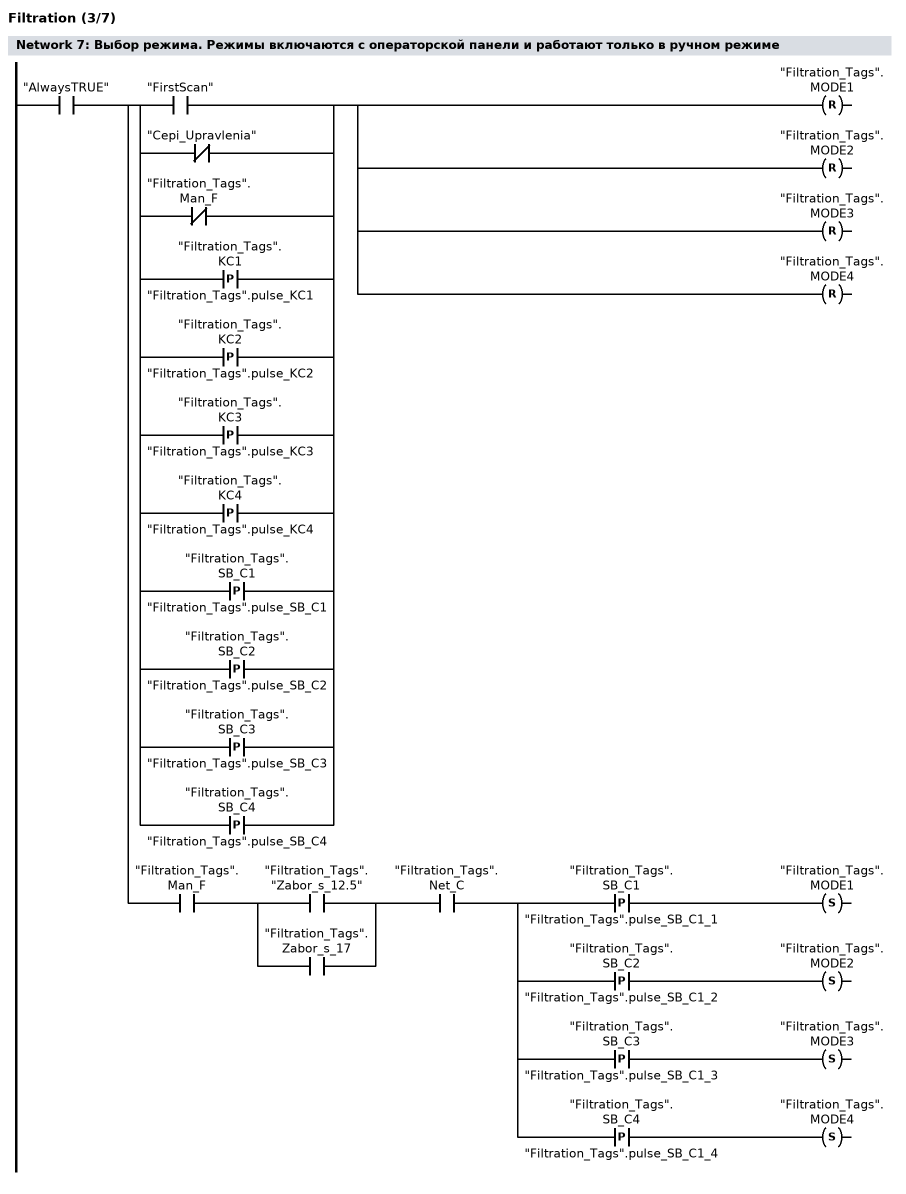
   RUNG wire#powerrail
      Contact( "AlwaysTRUE" )
      wire#w1
      Contact( "FirstScan" )
      wire#w2
      R_Coil( "Filtration_Tags".MODE1 )
   END_RUNG
   RUNG wire#w1
      I_Contact( "Cepi_Upravlenia" )
   END_RUNG wire#w2
   RUNG wire#w1
      I_Contact( "Filtration_Tags".Man_F )
   END_RUNG wire#w2
   RUNG wire#w1
      P_Contact(operand := "Filtration_Tags".KC1, bit := "Filtration_Tags".pulse_KC1)
   END_RUNG wire#w2
   RUNG wire#w1
      P_Contact(operand := "Filtration_Tags".KC2, bit := "Filtration_Tags".pulse_KC2)
   END_RUNG wire#w2
   RUNG wire#w1
      P_Contact(operand := "Filtration_Tags".KC3, bit := "Filtration_Tags".pulse_KC3)
   END_RUNG wire#w2
   RUNG wire#w1
      P_Contact(operand := "Filtration_Tags".KC4, bit := "Filtration_Tags".pulse_KC4)
   END_RUNG wire#w2
   RUNG wire#w1
      P_Contact(operand := "Filtration_Tags".SB_C1, bit := "Filtration_Tags".pulse_SB_C1)
   END_RUNG wire#w2
   RUNG wire#w1
      P_Contact(operand := "Filtration_Tags".SB_C2, bit := "Filtration_Tags".pulse_SB_C2)
   END_RUNG wire#w2
   RUNG wire#w1
      P_Contact(operand := "Filtration_Tags".SB_C3, bit := "Filtration_Tags".pulse_SB_C3)
   END_RUNG wire#w2
   RUNG wire#w1
      P_Contact(operand := "Filtration_Tags".SB_C4, bit := "Filtration_Tags".pulse_SB_C4)
   END_RUNG wire#w2
   RUNG wire#w2
      R_Coil( "Filtration_Tags".MODE2 )
   END_RUNG
   RUNG wire#w2
      R_Coil( "Filtration_Tags".MODE3 )
   END_RUNG
   RUNG wire#w2
      R_Coil( "Filtration_Tags".MODE4 )
   END_RUNG
   RUNG wire#w1
      Contact( "Filtration_Tags".Man_F )
      wire#w3
      Contact( "Filtration_Tags"."Zabor_s_12.5" )
      wire#w4
      Contact( "Filtration_Tags".Net_C )
      wire#w5
      P_Contact(operand := "Filtration_Tags".SB_C1, bit := "Filtration_Tags".pulse_SB_C1_1)
      S_Coil( "Filtration_Tags".MODE1 )
   END_RUNG
   RUNG wire#w3
      Contact( "Filtration_Tags".Zabor_s_17 )
   END_RUNG wire#w4
   RUNG wire#w5
      P_Contact(operand := "Filtration_Tags".SB_C2, bit := "Filtration_Tags".pulse_SB_C1_2)
      S_Coil( "Filtration_Tags".MODE2 )
   END_RUNG
   RUNG wire#w5
      P_Contact(operand := "Filtration_Tags".SB_C3, bit := "Filtration_Tags".pulse_SB_C1_3)
      S_Coil( "Filtration_Tags".MODE3 )
   END_RUNG
   RUNG wire#w5
      P_Contact(operand := "Filtration_Tags".SB_C4, bit := "Filtration_Tags".pulse_SB_C1_4)
      S_Coil( "Filtration_Tags".MODE4 )
   END_RUNG
   // the same network as SCL:
   #_w1 := "AlwaysTRUE" AND "Filtration_Tags".KC1 AND NOT "Filtration_Tags".pulse_KC1;   // rising edge of "Filtration_Tags".KC1
   "Filtration_Tags".pulse_KC1 := "Filtration_Tags".KC1;
   #_w2 := "AlwaysTRUE" AND "Filtration_Tags".KC2 AND NOT "Filtration_Tags".pulse_KC2;   // rising edge of "Filtration_Tags".KC2
   "Filtration_Tags".pulse_KC2 := "Filtration_Tags".KC2;
   #_w3 := "AlwaysTRUE" AND "Filtration_Tags".KC3 AND NOT "Filtration_Tags".pulse_KC3;   // rising edge of "Filtration_Tags".KC3
   "Filtration_Tags".pulse_KC3 := "Filtration_Tags".KC3;
   #_w4 := "AlwaysTRUE" AND "Filtration_Tags".KC4 AND NOT "Filtration_Tags".pulse_KC4;   // rising edge of "Filtration_Tags".KC4
   "Filtration_Tags".pulse_KC4 := "Filtration_Tags".KC4;
   #_w5 := "AlwaysTRUE" AND "Filtration_Tags".SB_C1 AND NOT "Filtration_Tags".pulse_SB_C1;   // rising edge of "Filtration_Tags".SB_C1
   "Filtration_Tags".pulse_SB_C1 := "Filtration_Tags".SB_C1;
   #_w6 := "AlwaysTRUE" AND "Filtration_Tags".SB_C2 AND NOT "Filtration_Tags".pulse_SB_C2;   // rising edge of "Filtration_Tags".SB_C2
   "Filtration_Tags".pulse_SB_C2 := "Filtration_Tags".SB_C2;
   #_w7 := "AlwaysTRUE" AND "Filtration_Tags".SB_C3 AND NOT "Filtration_Tags".pulse_SB_C3;   // rising edge of "Filtration_Tags".SB_C3
   "Filtration_Tags".pulse_SB_C3 := "Filtration_Tags".SB_C3;
   #_w8 := "AlwaysTRUE" AND "Filtration_Tags".SB_C4 AND NOT "Filtration_Tags".pulse_SB_C4;   // rising edge of "Filtration_Tags".SB_C4
   "Filtration_Tags".pulse_SB_C4 := "Filtration_Tags".SB_C4;
   IF ("AlwaysTRUE" AND ("FirstScan" OR NOT "Cepi_Upravlenia" OR NOT "Filtration_Tags".Man_F)) OR #_w1 OR #_w2 OR #_w3 OR #_w4 OR #_w5 OR #_w6 OR #_w7 OR #_w8 THEN
       "Filtration_Tags".MODE1 := FALSE;
       "Filtration_Tags".MODE2 := FALSE;
       "Filtration_Tags".MODE3 := FALSE;
       "Filtration_Tags".MODE4 := FALSE;
   END_IF;
   #_w9 := "AlwaysTRUE" AND "Filtration_Tags".Man_F AND ("Filtration_Tags"."Zabor_s_12.5" OR "Filtration_Tags".Zabor_s_17) AND "Filtration_Tags".Net_C;
   #_w10 := #_w9 AND "Filtration_Tags".SB_C1 AND NOT "Filtration_Tags".pulse_SB_C1_1;   // rising edge of "Filtration_Tags".SB_C1
   "Filtration_Tags".pulse_SB_C1_1 := "Filtration_Tags".SB_C1;
   IF #_w10 THEN "Filtration_Tags".MODE1 := TRUE; END_IF;
   #_w11 := #_w9 AND "Filtration_Tags".SB_C2 AND NOT "Filtration_Tags".pulse_SB_C1_2;   // rising edge of "Filtration_Tags".SB_C2
   "Filtration_Tags".pulse_SB_C1_2 := "Filtration_Tags".SB_C2;
   IF #_w11 THEN "Filtration_Tags".MODE2 := TRUE; END_IF;
   #_w12 := #_w9 AND "Filtration_Tags".SB_C3 AND NOT "Filtration_Tags".pulse_SB_C1_3;   // rising edge of "Filtration_Tags".SB_C3
   "Filtration_Tags".pulse_SB_C1_3 := "Filtration_Tags".SB_C3;
   IF #_w12 THEN "Filtration_Tags".MODE3 := TRUE; END_IF;
   #_w13 := #_w9 AND "Filtration_Tags".SB_C4 AND NOT "Filtration_Tags".pulse_SB_C1_4;   // rising edge of "Filtration_Tags".SB_C4
   "Filtration_Tags".pulse_SB_C1_4 := "Filtration_Tags".SB_C4;
   IF #_w13 THEN "Filtration_Tags".MODE4 := TRUE; END_IF;
END_REGION

REGION Network 8: Цикл 1. Заправка фильтра
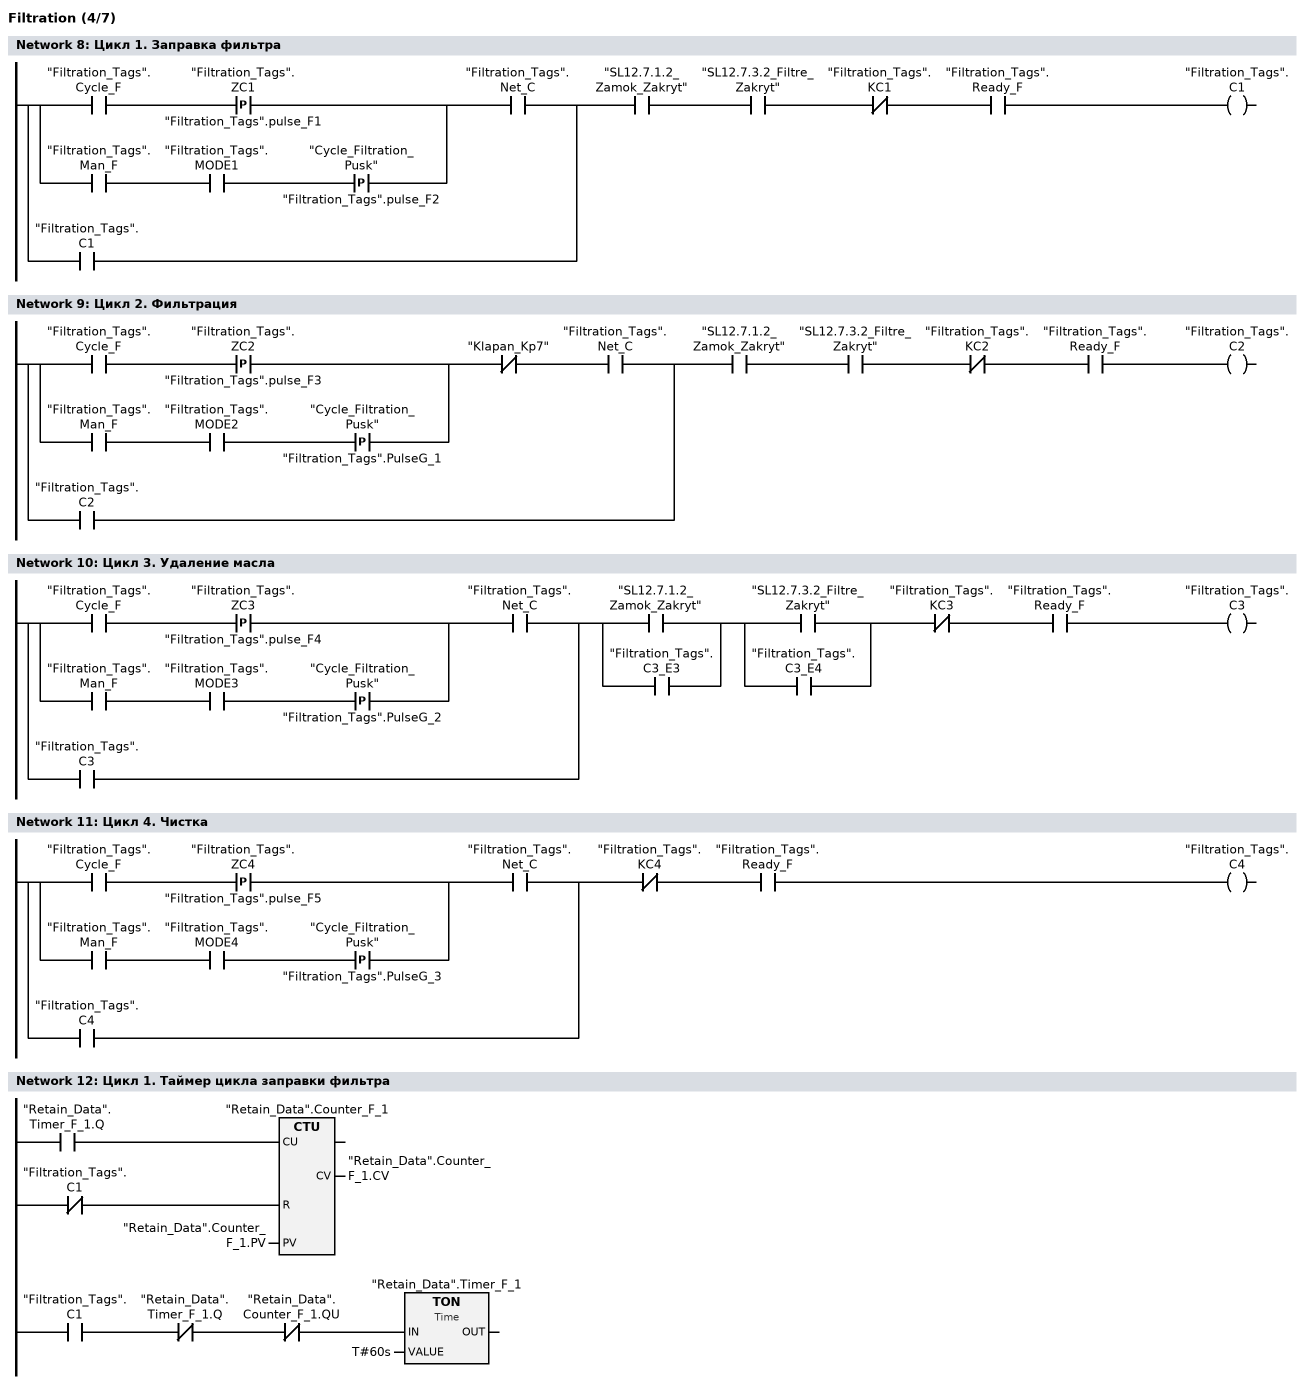
   RUNG wire#powerrail
      Contact( "Filtration_Tags".Cycle_F )
      P_Contact(operand := "Filtration_Tags".ZC1, bit := "Filtration_Tags".pulse_F1)
      wire#w1
      Contact( "Filtration_Tags".Net_C )
      wire#w2
      Contact( "SL12.7.1.2_Zamok_Zakryt" )
      Contact( "SL12.7.3.2_Filtre_Zakryt" )
      I_Contact( "Filtration_Tags".KC1 )
      Contact( "Filtration_Tags".Ready_F )
      Coil( "Filtration_Tags".C1 )
   END_RUNG
   RUNG wire#powerrail
      Contact( "Filtration_Tags".Man_F )
      Contact( "Filtration_Tags".MODE1 )
      P_Contact(operand := "Cycle_Filtration_Pusk", bit := "Filtration_Tags".pulse_F2)
   END_RUNG wire#w1
   RUNG wire#powerrail
      Contact( "Filtration_Tags".C1 )
   END_RUNG wire#w2
   // the same network as SCL:
   #_w1 := "Filtration_Tags".Cycle_F AND "Filtration_Tags".ZC1 AND NOT "Filtration_Tags".pulse_F1;   // rising edge of "Filtration_Tags".ZC1
   "Filtration_Tags".pulse_F1 := "Filtration_Tags".ZC1;
   #_w2 := "Filtration_Tags".Man_F AND "Filtration_Tags".MODE1 AND "Cycle_Filtration_Pusk" AND NOT "Filtration_Tags".pulse_F2;   // rising edge of "Cycle_Filtration_Pusk"
   "Filtration_Tags".pulse_F2 := "Cycle_Filtration_Pusk";
   "Filtration_Tags".C1 := (((#_w1 OR #_w2) AND "Filtration_Tags".Net_C) OR "Filtration_Tags".C1) AND "SL12.7.1.2_Zamok_Zakryt" AND "SL12.7.3.2_Filtre_Zakryt" AND NOT "Filtration_Tags".KC1 AND "Filtration_Tags".Ready_F;
END_REGION

REGION Network 9: Цикл 2. Фильтрация
   RUNG wire#powerrail
      Contact( "Filtration_Tags".Cycle_F )
      P_Contact(operand := "Filtration_Tags".ZC2, bit := "Filtration_Tags".pulse_F3)
      wire#w1
      I_Contact( "Klapan_Kp7" )
      Contact( "Filtration_Tags".Net_C )
      wire#w2
      Contact( "SL12.7.1.2_Zamok_Zakryt" )
      Contact( "SL12.7.3.2_Filtre_Zakryt" )
      I_Contact( "Filtration_Tags".KC2 )
      Contact( "Filtration_Tags".Ready_F )
      Coil( "Filtration_Tags".C2 )
   END_RUNG
   RUNG wire#powerrail
      Contact( "Filtration_Tags".Man_F )
      Contact( "Filtration_Tags".MODE2 )
      P_Contact(operand := "Cycle_Filtration_Pusk", bit := "Filtration_Tags".PulseG_1)
   END_RUNG wire#w1
   RUNG wire#powerrail
      Contact( "Filtration_Tags".C2 )
   END_RUNG wire#w2
   // the same network as SCL:
   #_w1 := "Filtration_Tags".Cycle_F AND "Filtration_Tags".ZC2 AND NOT "Filtration_Tags".pulse_F3;   // rising edge of "Filtration_Tags".ZC2
   "Filtration_Tags".pulse_F3 := "Filtration_Tags".ZC2;
   #_w2 := "Filtration_Tags".Man_F AND "Filtration_Tags".MODE2 AND "Cycle_Filtration_Pusk" AND NOT "Filtration_Tags".PulseG_1;   // rising edge of "Cycle_Filtration_Pusk"
   "Filtration_Tags".PulseG_1 := "Cycle_Filtration_Pusk";
   "Filtration_Tags".C2 := (((#_w1 OR #_w2) AND NOT "Klapan_Kp7" AND "Filtration_Tags".Net_C) OR "Filtration_Tags".C2) AND "SL12.7.1.2_Zamok_Zakryt" AND "SL12.7.3.2_Filtre_Zakryt" AND NOT "Filtration_Tags".KC2 AND "Filtration_Tags".Ready_F;
END_REGION

REGION Network 10: Цикл 3. Удаление масла
   RUNG wire#powerrail
      Contact( "Filtration_Tags".Cycle_F )
      P_Contact(operand := "Filtration_Tags".ZC3, bit := "Filtration_Tags".pulse_F4)
      wire#w1
      Contact( "Filtration_Tags".Net_C )
      wire#w2
      Contact( "SL12.7.1.2_Zamok_Zakryt" )
      wire#w3
      Contact( "SL12.7.3.2_Filtre_Zakryt" )
      wire#w4
      I_Contact( "Filtration_Tags".KC3 )
      Contact( "Filtration_Tags".Ready_F )
      Coil( "Filtration_Tags".C3 )
   END_RUNG
   RUNG wire#powerrail
      Contact( "Filtration_Tags".Man_F )
      Contact( "Filtration_Tags".MODE3 )
      P_Contact(operand := "Cycle_Filtration_Pusk", bit := "Filtration_Tags".PulseG_2)
   END_RUNG wire#w1
   RUNG wire#powerrail
      Contact( "Filtration_Tags".C3 )
   END_RUNG wire#w2
   RUNG wire#w2
      Contact( "Filtration_Tags".C3_E3 )
   END_RUNG wire#w3
   RUNG wire#w3
      Contact( "Filtration_Tags".C3_E4 )
   END_RUNG wire#w4
   // the same network as SCL:
   #_w1 := "Filtration_Tags".Cycle_F AND "Filtration_Tags".ZC3 AND NOT "Filtration_Tags".pulse_F4;   // rising edge of "Filtration_Tags".ZC3
   "Filtration_Tags".pulse_F4 := "Filtration_Tags".ZC3;
   #_w2 := "Filtration_Tags".Man_F AND "Filtration_Tags".MODE3 AND "Cycle_Filtration_Pusk" AND NOT "Filtration_Tags".PulseG_2;   // rising edge of "Cycle_Filtration_Pusk"
   "Filtration_Tags".PulseG_2 := "Cycle_Filtration_Pusk";
   "Filtration_Tags".C3 := (((#_w1 OR #_w2) AND "Filtration_Tags".Net_C) OR "Filtration_Tags".C3) AND ("SL12.7.1.2_Zamok_Zakryt" OR "Filtration_Tags".C3_E3) AND ("SL12.7.3.2_Filtre_Zakryt" OR "Filtration_Tags".C3_E4) AND NOT "Filtration_Tags".KC3 AND "Filtration_Tags".Ready_F;
END_REGION

REGION Network 11: Цикл 4. Чистка
   RUNG wire#powerrail
      Contact( "Filtration_Tags".Cycle_F )
      P_Contact(operand := "Filtration_Tags".ZC4, bit := "Filtration_Tags".pulse_F5)
      wire#w1
      Contact( "Filtration_Tags".Net_C )
      wire#w2
      I_Contact( "Filtration_Tags".KC4 )
      Contact( "Filtration_Tags".Ready_F )
      Coil( "Filtration_Tags".C4 )
   END_RUNG
   RUNG wire#powerrail
      Contact( "Filtration_Tags".Man_F )
      Contact( "Filtration_Tags".MODE4 )
      P_Contact(operand := "Cycle_Filtration_Pusk", bit := "Filtration_Tags".PulseG_3)
   END_RUNG wire#w1
   RUNG wire#powerrail
      Contact( "Filtration_Tags".C4 )
   END_RUNG wire#w2
   // the same network as SCL:
   #_w1 := "Filtration_Tags".Cycle_F AND "Filtration_Tags".ZC4 AND NOT "Filtration_Tags".pulse_F5;   // rising edge of "Filtration_Tags".ZC4
   "Filtration_Tags".pulse_F5 := "Filtration_Tags".ZC4;
   #_w2 := "Filtration_Tags".Man_F AND "Filtration_Tags".MODE4 AND "Cycle_Filtration_Pusk" AND NOT "Filtration_Tags".PulseG_3;   // rising edge of "Cycle_Filtration_Pusk"
   "Filtration_Tags".PulseG_3 := "Cycle_Filtration_Pusk";
   "Filtration_Tags".C4 := (((#_w1 OR #_w2) AND "Filtration_Tags".Net_C) OR "Filtration_Tags".C4) AND NOT "Filtration_Tags".KC4 AND "Filtration_Tags".Ready_F;
END_REGION

REGION Network 12: Цикл 1. Таймер цикла заправки фильтра
   "Retain_Data".Counter_F_1.CTU(CU := "Retain_Data".Timer_F_1.Q,
                           R := NOT "Filtration_Tags".C1,
                           PV := "Retain_Data".Counter_F_1.PV,
                           CV => "Retain_Data".Counter_F_1.CV);
   "Retain_Data".Timer_F_1.TON(IN := "Filtration_Tags".C1 AND NOT "Retain_Data".Timer_F_1.Q AND NOT "Retain_Data".Counter_F_1.QU, PT := T#60s);   // TON coil
END_REGION

REGION Network 13: Цикл 1. Таймер работы клапана декомпрессии Кд
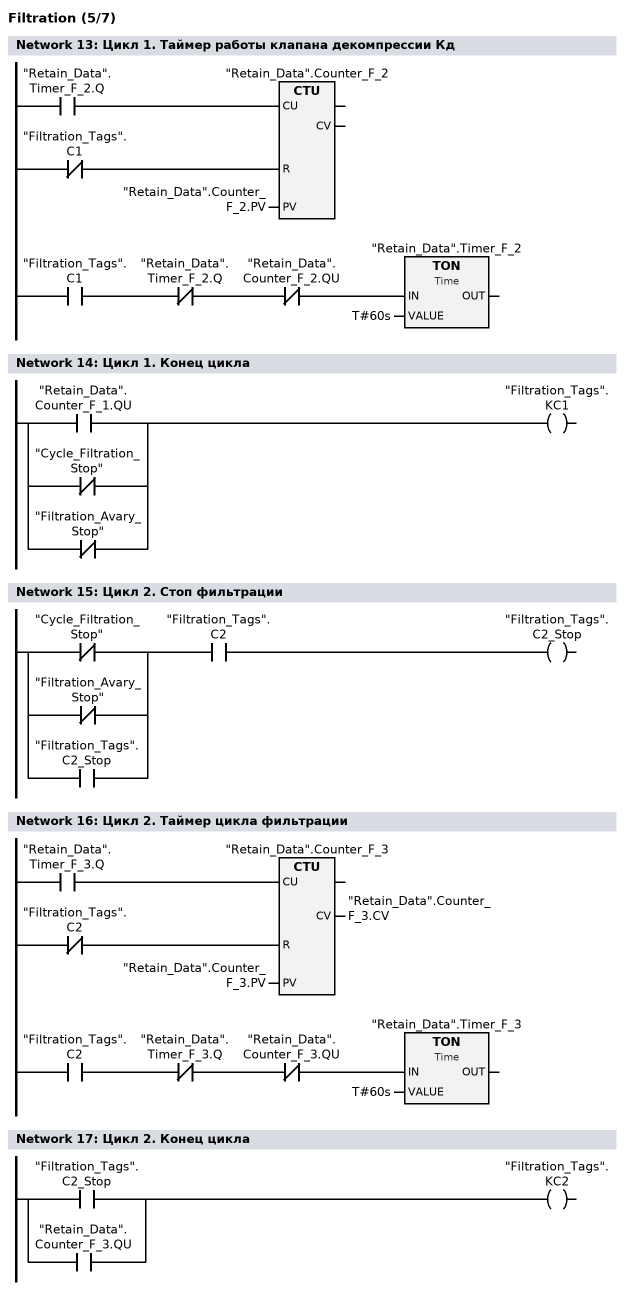
   "Retain_Data".Counter_F_2.CTU(CU := "Retain_Data".Timer_F_2.Q,
                           R := NOT "Filtration_Tags".C1,
                           PV := "Retain_Data".Counter_F_2.PV);
   "Retain_Data".Timer_F_2.TON(IN := "Filtration_Tags".C1 AND NOT "Retain_Data".Timer_F_2.Q AND NOT "Retain_Data".Counter_F_2.QU, PT := T#60s);   // TON coil
END_REGION

REGION Network 14: Цикл 1. Конец цикла
   RUNG wire#powerrail
      Contact( "Retain_Data".Counter_F_1.QU )
      wire#w1
      Coil( "Filtration_Tags".KC1 )
   END_RUNG
   RUNG wire#powerrail
      I_Contact( "Cycle_Filtration_Stop" )
   END_RUNG wire#w1
   RUNG wire#powerrail
      I_Contact( "Filtration_Avary_Stop" )
   END_RUNG wire#w1
   // the same network as SCL:
   "Filtration_Tags".KC1 := "Retain_Data".Counter_F_1.QU OR NOT "Cycle_Filtration_Stop" OR NOT "Filtration_Avary_Stop";
END_REGION

REGION Network 15: Цикл 2. Стоп фильтрации
   RUNG wire#powerrail
      I_Contact( "Cycle_Filtration_Stop" )
      wire#w1
      Contact( "Filtration_Tags".C2 )
      Coil( "Filtration_Tags".C2_Stop )
   END_RUNG
   RUNG wire#powerrail
      I_Contact( "Filtration_Avary_Stop" )
   END_RUNG wire#w1
   RUNG wire#powerrail
      Contact( "Filtration_Tags".C2_Stop )
   END_RUNG wire#w1
   // the same network as SCL:
   "Filtration_Tags".C2_Stop := (NOT "Cycle_Filtration_Stop" OR NOT "Filtration_Avary_Stop" OR "Filtration_Tags".C2_Stop) AND "Filtration_Tags".C2;
END_REGION

REGION Network 16: Цикл 2. Таймер цикла фильтрации
   "Retain_Data".Counter_F_3.CTU(CU := "Retain_Data".Timer_F_3.Q,
                           R := NOT "Filtration_Tags".C2,
                           PV := "Retain_Data".Counter_F_3.PV,
                           CV => "Retain_Data".Counter_F_3.CV);
   "Retain_Data".Timer_F_3.TON(IN := "Filtration_Tags".C2 AND NOT "Retain_Data".Timer_F_3.Q AND NOT "Retain_Data".Counter_F_3.QU, PT := T#60s);   // TON coil
END_REGION

REGION Network 17: Цикл 2. Конец цикла
   RUNG wire#powerrail
      Contact( "Filtration_Tags".C2_Stop )
      wire#w1
      Coil( "Filtration_Tags".KC2 )
   END_RUNG
   RUNG wire#powerrail
      Contact( "Retain_Data".Counter_F_3.QU )
   END_RUNG wire#w1
   // the same network as SCL:
   "Filtration_Tags".KC2 := "Filtration_Tags".C2_Stop OR "Retain_Data".Counter_F_3.QU;
END_REGION

REGION Network 18: Цикл 3. Циклограмма удаления масла
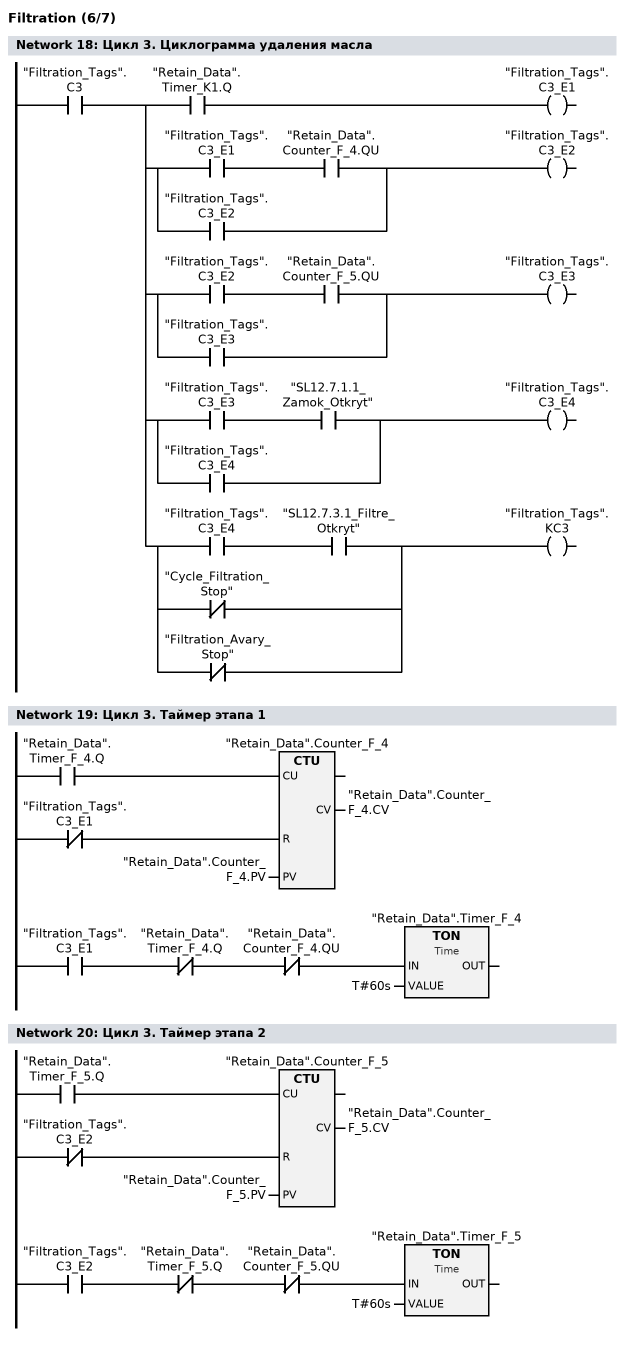
   RUNG wire#powerrail
      Contact( "Filtration_Tags".C3 )
      wire#w1
      Contact( "Retain_Data".Timer_K1.Q )
      Coil( "Filtration_Tags".C3_E1 )
   END_RUNG
   RUNG wire#w1
      Contact( "Filtration_Tags".C3_E1 )
      Contact( "Retain_Data".Counter_F_4.QU )
      wire#w2
      Coil( "Filtration_Tags".C3_E2 )
   END_RUNG
   RUNG wire#w1
      Contact( "Filtration_Tags".C3_E2 )
   END_RUNG wire#w2
   RUNG wire#w1
      Contact( "Filtration_Tags".C3_E2 )
      Contact( "Retain_Data".Counter_F_5.QU )
      wire#w3
      Coil( "Filtration_Tags".C3_E3 )
   END_RUNG
   RUNG wire#w1
      Contact( "Filtration_Tags".C3_E3 )
   END_RUNG wire#w3
   RUNG wire#w1
      Contact( "Filtration_Tags".C3_E3 )
      Contact( "SL12.7.1.1_Zamok_Otkryt" )
      wire#w4
      Coil( "Filtration_Tags".C3_E4 )
   END_RUNG
   RUNG wire#w1
      Contact( "Filtration_Tags".C3_E4 )
   END_RUNG wire#w4
   RUNG wire#w1
      Contact( "Filtration_Tags".C3_E4 )
      Contact( "SL12.7.3.1_Filtre_Otkryt" )
      wire#w5
      Coil( "Filtration_Tags".KC3 )
   END_RUNG
   RUNG wire#w1
      I_Contact( "Cycle_Filtration_Stop" )
   END_RUNG wire#w5
   RUNG wire#w1
      I_Contact( "Filtration_Avary_Stop" )
   END_RUNG wire#w5
   // the same network as SCL:
   "Filtration_Tags".C3_E1 := "Filtration_Tags".C3 AND "Retain_Data".Timer_K1.Q;
   "Filtration_Tags".C3_E2 := "Filtration_Tags".C3 AND (("Filtration_Tags".C3_E1 AND "Retain_Data".Counter_F_4.QU) OR "Filtration_Tags".C3_E2);
   "Filtration_Tags".C3_E3 := "Filtration_Tags".C3 AND (("Filtration_Tags".C3_E2 AND "Retain_Data".Counter_F_5.QU) OR "Filtration_Tags".C3_E3);
   "Filtration_Tags".C3_E4 := "Filtration_Tags".C3 AND (("Filtration_Tags".C3_E3 AND "SL12.7.1.1_Zamok_Otkryt") OR "Filtration_Tags".C3_E4);
   "Filtration_Tags".KC3 := "Filtration_Tags".C3 AND (("Filtration_Tags".C3_E4 AND "SL12.7.3.1_Filtre_Otkryt") OR NOT "Cycle_Filtration_Stop" OR NOT "Filtration_Avary_Stop");
END_REGION

REGION Network 19: Цикл 3. Таймер этапа 1
   "Retain_Data".Counter_F_4.CTU(CU := "Retain_Data".Timer_F_4.Q,
                           R := NOT "Filtration_Tags".C3_E1,
                           PV := "Retain_Data".Counter_F_4.PV,
                           CV => "Retain_Data".Counter_F_4.CV);
   "Retain_Data".Timer_F_4.TON(IN := "Filtration_Tags".C3_E1 AND NOT "Retain_Data".Timer_F_4.Q AND NOT "Retain_Data".Counter_F_4.QU, PT := T#60s);   // TON coil
END_REGION

REGION Network 20: Цикл 3. Таймер этапа 2
   "Retain_Data".Counter_F_5.CTU(CU := "Retain_Data".Timer_F_5.Q,
                           R := NOT "Filtration_Tags".C3_E2,
                           PV := "Retain_Data".Counter_F_5.PV,
                           CV => "Retain_Data".Counter_F_5.CV);
   "Retain_Data".Timer_F_5.TON(IN := "Filtration_Tags".C3_E2 AND NOT "Retain_Data".Timer_F_5.Q AND NOT "Retain_Data".Counter_F_5.QU, PT := T#60s);   // TON coil
END_REGION

REGION Network 21: Цикл 4. Циклограмма чистки
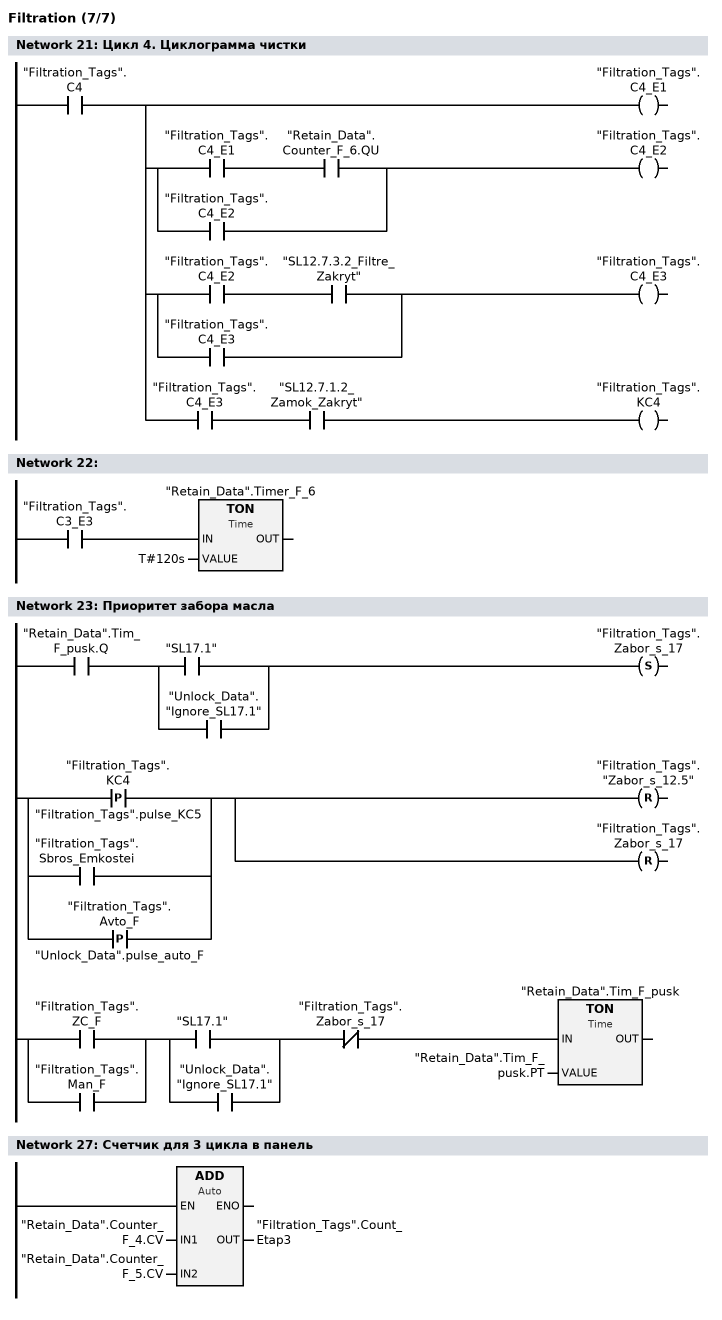
   RUNG wire#powerrail
      Contact( "Filtration_Tags".C4 )
      wire#w1
      Coil( "Filtration_Tags".C4_E1 )
   END_RUNG
   RUNG wire#w1
      Contact( "Filtration_Tags".C4_E1 )
      Contact( "Retain_Data".Counter_F_6.QU )
      wire#w2
      Coil( "Filtration_Tags".C4_E2 )
   END_RUNG
   RUNG wire#w1
      Contact( "Filtration_Tags".C4_E2 )
   END_RUNG wire#w2
   RUNG wire#w1
      Contact( "Filtration_Tags".C4_E2 )
      Contact( "SL12.7.3.2_Filtre_Zakryt" )
      wire#w3
      Coil( "Filtration_Tags".C4_E3 )
   END_RUNG
   RUNG wire#w1
      Contact( "Filtration_Tags".C4_E3 )
   END_RUNG wire#w3
   RUNG wire#w1
      Contact( "Filtration_Tags".C4_E3 )
      Contact( "SL12.7.1.2_Zamok_Zakryt" )
      Coil( "Filtration_Tags".KC4 )
   END_RUNG
   // the same network as SCL:
   "Filtration_Tags".C4_E1 := "Filtration_Tags".C4;
   "Filtration_Tags".C4_E2 := "Filtration_Tags".C4 AND (("Filtration_Tags".C4_E1 AND "Retain_Data".Counter_F_6.QU) OR "Filtration_Tags".C4_E2);
   "Filtration_Tags".C4_E3 := "Filtration_Tags".C4 AND (("Filtration_Tags".C4_E2 AND "SL12.7.3.2_Filtre_Zakryt") OR "Filtration_Tags".C4_E3);
   "Filtration_Tags".KC4 := "Filtration_Tags".C4 AND "Filtration_Tags".C4_E3 AND "SL12.7.1.2_Zamok_Zakryt";
END_REGION

REGION Network 22
   "Retain_Data".Timer_F_6.TON(IN := "Filtration_Tags".C3_E3, PT := T#120s);   // TON coil
END_REGION

REGION Network 23: Приоритет забора масла
   IF "Retain_Data".Tim_F_pusk.Q AND ("SL17.1" OR "Unlock_Data"."Ignore_SL17.1") THEN
       "Filtration_Tags".Zabor_s_17 := TRUE;
   END_IF;
   #_w1 := "Filtration_Tags".KC4 AND NOT "Filtration_Tags".pulse_KC5;   // rising edge of "Filtration_Tags".KC4
   "Filtration_Tags".pulse_KC5 := "Filtration_Tags".KC4;
   #_w2 := "Filtration_Tags".Avto_F AND NOT "Unlock_Data".pulse_auto_F;   // rising edge of "Filtration_Tags".Avto_F
   "Unlock_Data".pulse_auto_F := "Filtration_Tags".Avto_F;
   IF #_w1 OR "Filtration_Tags".Sbros_Emkostei OR #_w2 THEN
       "Filtration_Tags"."Zabor_s_12.5" := FALSE;
       "Filtration_Tags".Zabor_s_17 := FALSE;
   END_IF;
   "Retain_Data".Tim_F_pusk.TON(IN := ("Filtration_Tags".ZC_F OR "Filtration_Tags".Man_F) AND ("SL17.1" OR "Unlock_Data"."Ignore_SL17.1") AND NOT "Filtration_Tags".Zabor_s_17, PT := "Retain_Data".Tim_F_pusk.PT);   // TON coil
END_REGION

REGION Network 24: Работа насоса М19Н
END_REGION

REGION Network 25: Ошибка переполнения емкостей 22.1 и 22.2
END_REGION

REGION Network 26: Бит отвеса для W2
END_REGION

REGION Network 27: Счетчик для 3 цикла в панель
   RUNG wire#powerrail
      Add(in1 := "Retain_Data".Counter_F_4.CV, in2 := "Retain_Data".Counter_F_5.CV, out => "Filtration_Tags".Count_Etap3)
   END_RUNG
   // the same network as SCL:
   "Filtration_Tags".Count_Etap3 := "Retain_Data".Counter_F_4.CV + "Retain_Data".Counter_F_5.CV;
END_REGION
END_FUNCTION_BLOCK

FUNCTION_BLOCK "Motors_F"   // FB6, LAD
{ S7_Optimized_Access := 'TRUE' }
VERSION : 0.1
   VAR_TEMP   // added for the SCL form of the ladder/FBD networks
      _w1 : Bool;
   END_VAR
BEGIN

REGION Network 1: Клапан К1
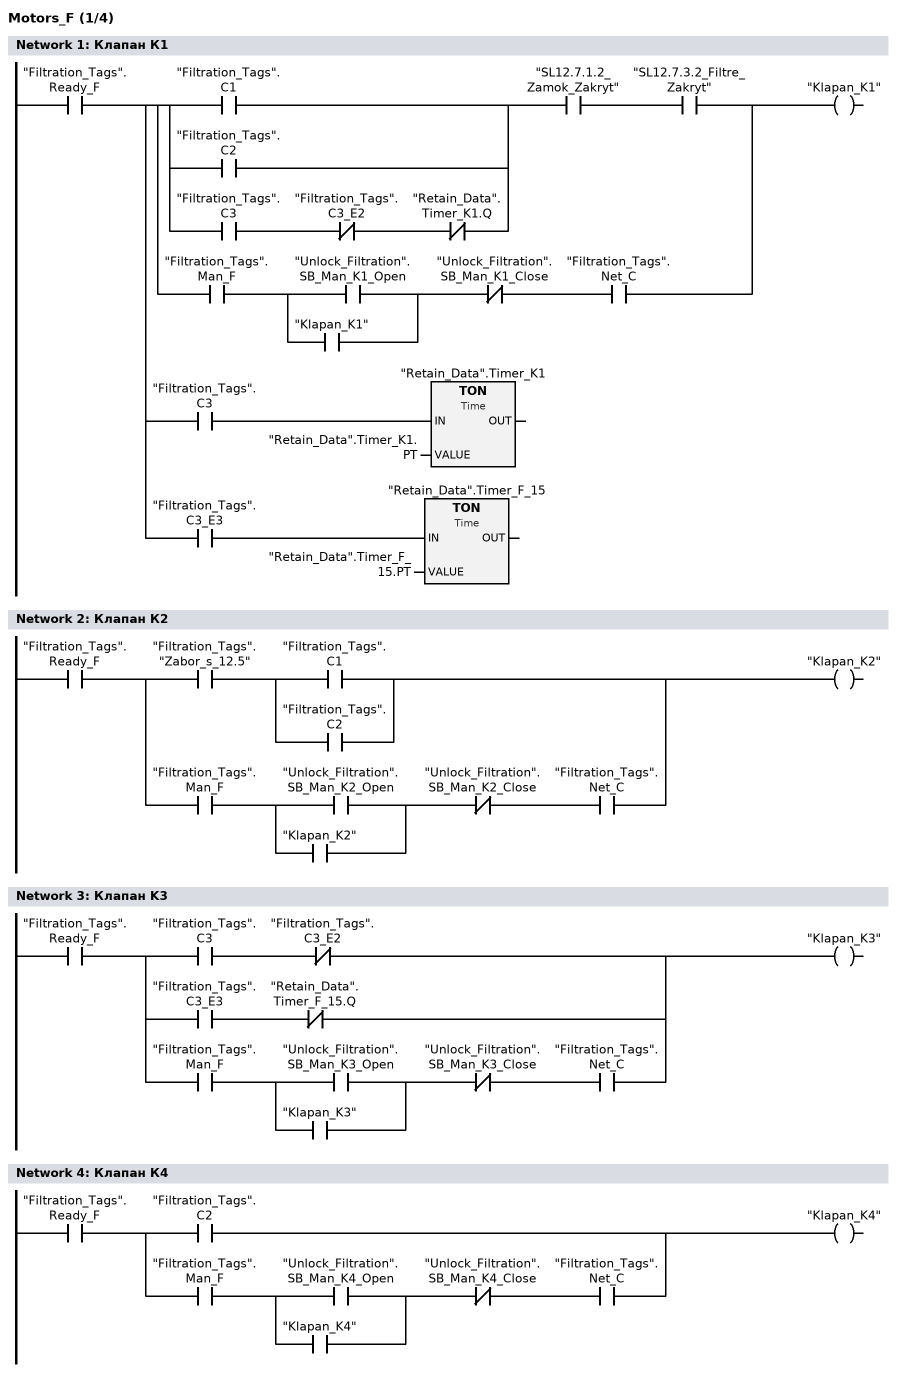
   "Klapan_K1" := "Filtration_Tags".Ready_F AND ((("Filtration_Tags".C1 OR "Filtration_Tags".C2 OR ("Filtration_Tags".C3 AND NOT "Filtration_Tags".C3_E2 AND NOT "Retain_Data".Timer_K1.Q)) AND "SL12.7.1.2_Zamok_Zakryt" AND "SL12.7.3.2_Filtre_Zakryt") OR ("Filtration_Tags".Man_F AND ("Unlock_Filtration".SB_Man_K1_Open OR "Klapan_K1") AND NOT "Unlock_Filtration".SB_Man_K1_Close AND "Filtration_Tags".Net_C));
   "Retain_Data".Timer_K1.TON(IN := "Filtration_Tags".Ready_F AND "Filtration_Tags".C3, PT := "Retain_Data".Timer_K1.PT);   // TON coil
   "Retain_Data".Timer_F_15.TON(IN := "Filtration_Tags".Ready_F AND "Filtration_Tags".C3_E3, PT := "Retain_Data".Timer_F_15.PT);   // TON coil
END_REGION

REGION Network 2: Клапан К2
   RUNG wire#powerrail
      Contact( "Filtration_Tags".Ready_F )
      wire#w1
      Contact( "Filtration_Tags"."Zabor_s_12.5" )
      wire#w2
      Contact( "Filtration_Tags".C1 )
      wire#w3
      Coil( "Klapan_K2" )
   END_RUNG
   RUNG wire#w2
      Contact( "Filtration_Tags".C2 )
   END_RUNG wire#w3
   RUNG wire#w1
      Contact( "Filtration_Tags".Man_F )
      wire#w4
      Contact( "Unlock_Filtration".SB_Man_K2_Open )
      wire#w5
      I_Contact( "Unlock_Filtration".SB_Man_K2_Close )
      Contact( "Filtration_Tags".Net_C )
   END_RUNG wire#w3
   RUNG wire#w4
      Contact( "Klapan_K2" )
   END_RUNG wire#w5
   // the same network as SCL:
   "Klapan_K2" := "Filtration_Tags".Ready_F AND (("Filtration_Tags"."Zabor_s_12.5" AND ("Filtration_Tags".C1 OR "Filtration_Tags".C2)) OR ("Filtration_Tags".Man_F AND ("Unlock_Filtration".SB_Man_K2_Open OR "Klapan_K2") AND NOT "Unlock_Filtration".SB_Man_K2_Close AND "Filtration_Tags".Net_C));
END_REGION

REGION Network 3: Клапан K3
   RUNG wire#powerrail
      Contact( "Filtration_Tags".Ready_F )
      wire#w1
      Contact( "Filtration_Tags".C3 )
      I_Contact( "Filtration_Tags".C3_E2 )
      wire#w2
      Coil( "Klapan_K3" )
   END_RUNG
   RUNG wire#w1
      Contact( "Filtration_Tags".C3_E3 )
      I_Contact( "Retain_Data".Timer_F_15.Q )
   END_RUNG wire#w2
   RUNG wire#w1
      Contact( "Filtration_Tags".Man_F )
      wire#w3
      Contact( "Unlock_Filtration".SB_Man_K3_Open )
      wire#w4
      I_Contact( "Unlock_Filtration".SB_Man_K3_Close )
      Contact( "Filtration_Tags".Net_C )
   END_RUNG wire#w2
   RUNG wire#w3
      Contact( "Klapan_K3" )
   END_RUNG wire#w4
   // the same network as SCL:
   "Klapan_K3" := "Filtration_Tags".Ready_F AND (("Filtration_Tags".C3 AND NOT "Filtration_Tags".C3_E2) OR ("Filtration_Tags".C3_E3 AND NOT "Retain_Data".Timer_F_15.Q) OR ("Filtration_Tags".Man_F AND ("Unlock_Filtration".SB_Man_K3_Open OR "Klapan_K3") AND NOT "Unlock_Filtration".SB_Man_K3_Close AND "Filtration_Tags".Net_C));
END_REGION

REGION Network 4: Клапан К4
   RUNG wire#powerrail
      Contact( "Filtration_Tags".Ready_F )
      wire#w1
      Contact( "Filtration_Tags".C2 )
      wire#w2
      Coil( "Klapan_K4" )
   END_RUNG
   RUNG wire#w1
      Contact( "Filtration_Tags".Man_F )
      wire#w3
      Contact( "Unlock_Filtration".SB_Man_K4_Open )
      wire#w4
      I_Contact( "Unlock_Filtration".SB_Man_K4_Close )
      Contact( "Filtration_Tags".Net_C )
   END_RUNG wire#w2
   RUNG wire#w3
      Contact( "Klapan_K4" )
   END_RUNG wire#w4
   // the same network as SCL:
   "Klapan_K4" := "Filtration_Tags".Ready_F AND ("Filtration_Tags".C2 OR ("Filtration_Tags".Man_F AND ("Unlock_Filtration".SB_Man_K4_Open OR "Klapan_K4") AND NOT "Unlock_Filtration".SB_Man_K4_Close AND "Filtration_Tags".Net_C));
END_REGION

REGION Network 5: Клапан декомпрессии Кд
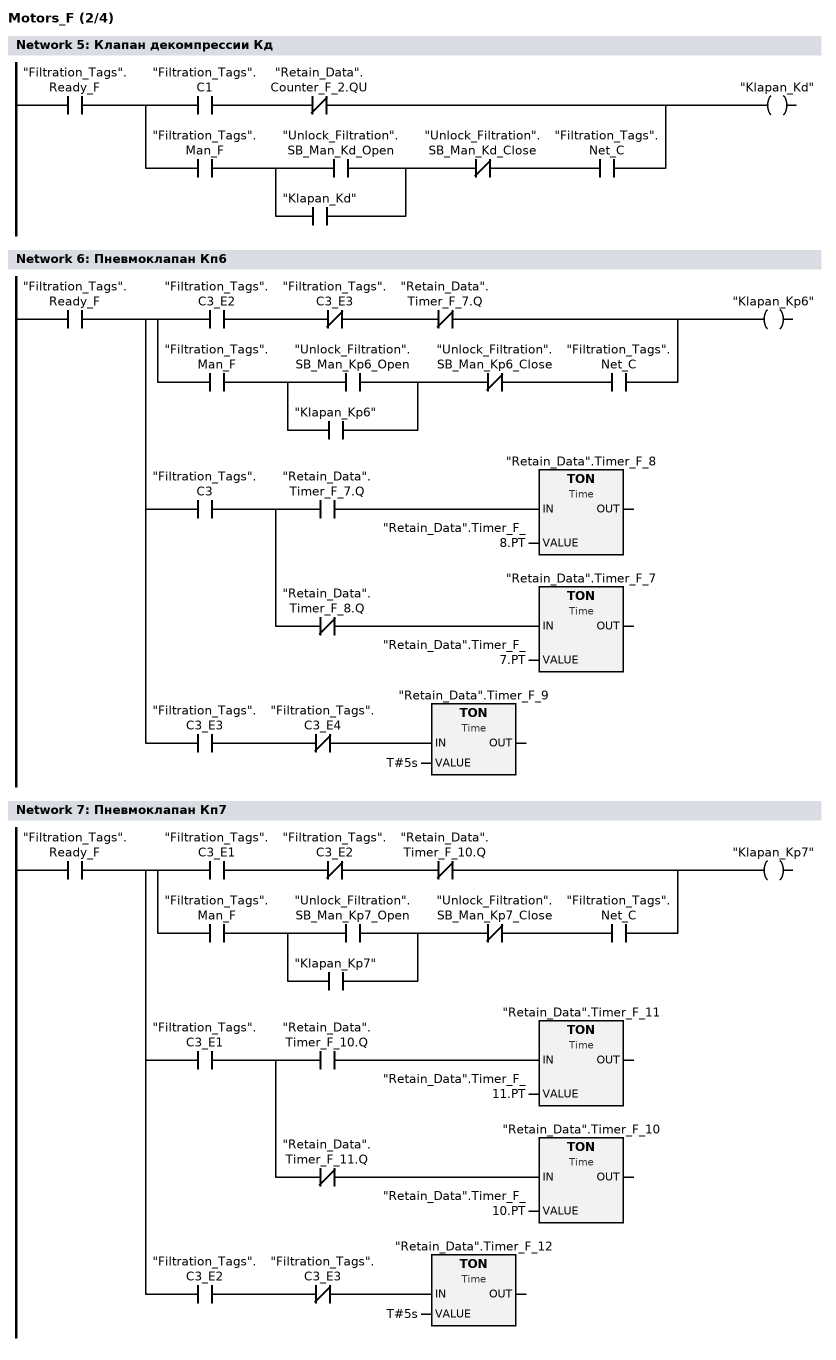
   RUNG wire#powerrail
      Contact( "Filtration_Tags".Ready_F )
      wire#w1
      Contact( "Filtration_Tags".C1 )
      I_Contact( "Retain_Data".Counter_F_2.QU )
      wire#w2
      Coil( "Klapan_Kd" )
   END_RUNG
   RUNG wire#w1
      Contact( "Filtration_Tags".Man_F )
      wire#w3
      Contact( "Unlock_Filtration".SB_Man_Kd_Open )
      wire#w4
      I_Contact( "Unlock_Filtration".SB_Man_Kd_Close )
      Contact( "Filtration_Tags".Net_C )
   END_RUNG wire#w2
   RUNG wire#w3
      Contact( "Klapan_Kd" )
   END_RUNG wire#w4
   // the same network as SCL:
   "Klapan_Kd" := "Filtration_Tags".Ready_F AND (("Filtration_Tags".C1 AND NOT "Retain_Data".Counter_F_2.QU) OR ("Filtration_Tags".Man_F AND ("Unlock_Filtration".SB_Man_Kd_Open OR "Klapan_Kd") AND NOT "Unlock_Filtration".SB_Man_Kd_Close AND "Filtration_Tags".Net_C));
END_REGION

REGION Network 6: Пневмоклапан Кп6
   "Klapan_Kp6" := "Filtration_Tags".Ready_F AND (("Filtration_Tags".C3_E2 AND NOT "Filtration_Tags".C3_E3 AND NOT "Retain_Data".Timer_F_7.Q) OR ("Filtration_Tags".Man_F AND ("Unlock_Filtration".SB_Man_Kp6_Open OR "Klapan_Kp6") AND NOT "Unlock_Filtration".SB_Man_Kp6_Close AND "Filtration_Tags".Net_C));
   #_w1 := "Filtration_Tags".Ready_F AND "Filtration_Tags".C3;
   "Retain_Data".Timer_F_8.TON(IN := #_w1 AND "Retain_Data".Timer_F_7.Q, PT := "Retain_Data".Timer_F_8.PT);   // TON coil
   "Retain_Data".Timer_F_7.TON(IN := #_w1 AND NOT "Retain_Data".Timer_F_8.Q, PT := "Retain_Data".Timer_F_7.PT);   // TON coil
   "Retain_Data".Timer_F_9.TON(IN := "Filtration_Tags".Ready_F AND "Filtration_Tags".C3_E3 AND NOT "Filtration_Tags".C3_E4, PT := T#5s);   // TON coil
END_REGION

REGION Network 7: Пневмоклапан Кп7
   "Klapan_Kp7" := "Filtration_Tags".Ready_F AND (("Filtration_Tags".C3_E1 AND NOT "Filtration_Tags".C3_E2 AND NOT "Retain_Data".Timer_F_10.Q) OR ("Filtration_Tags".Man_F AND ("Unlock_Filtration".SB_Man_Kp7_Open OR "Klapan_Kp7") AND NOT "Unlock_Filtration".SB_Man_Kp7_Close AND "Filtration_Tags".Net_C));
   #_w1 := "Filtration_Tags".Ready_F AND "Filtration_Tags".C3_E1;
   "Retain_Data".Timer_F_11.TON(IN := #_w1 AND "Retain_Data".Timer_F_10.Q, PT := "Retain_Data".Timer_F_11.PT);   // TON coil
   "Retain_Data".Timer_F_10.TON(IN := #_w1 AND NOT "Retain_Data".Timer_F_11.Q, PT := "Retain_Data".Timer_F_10.PT);   // TON coil
   "Retain_Data".Timer_F_12.TON(IN := "Filtration_Tags".Ready_F AND "Filtration_Tags".C3_E2 AND NOT "Filtration_Tags".C3_E3, PT := T#5s);   // TON coil
END_REGION

REGION Network 8: Вибромотор
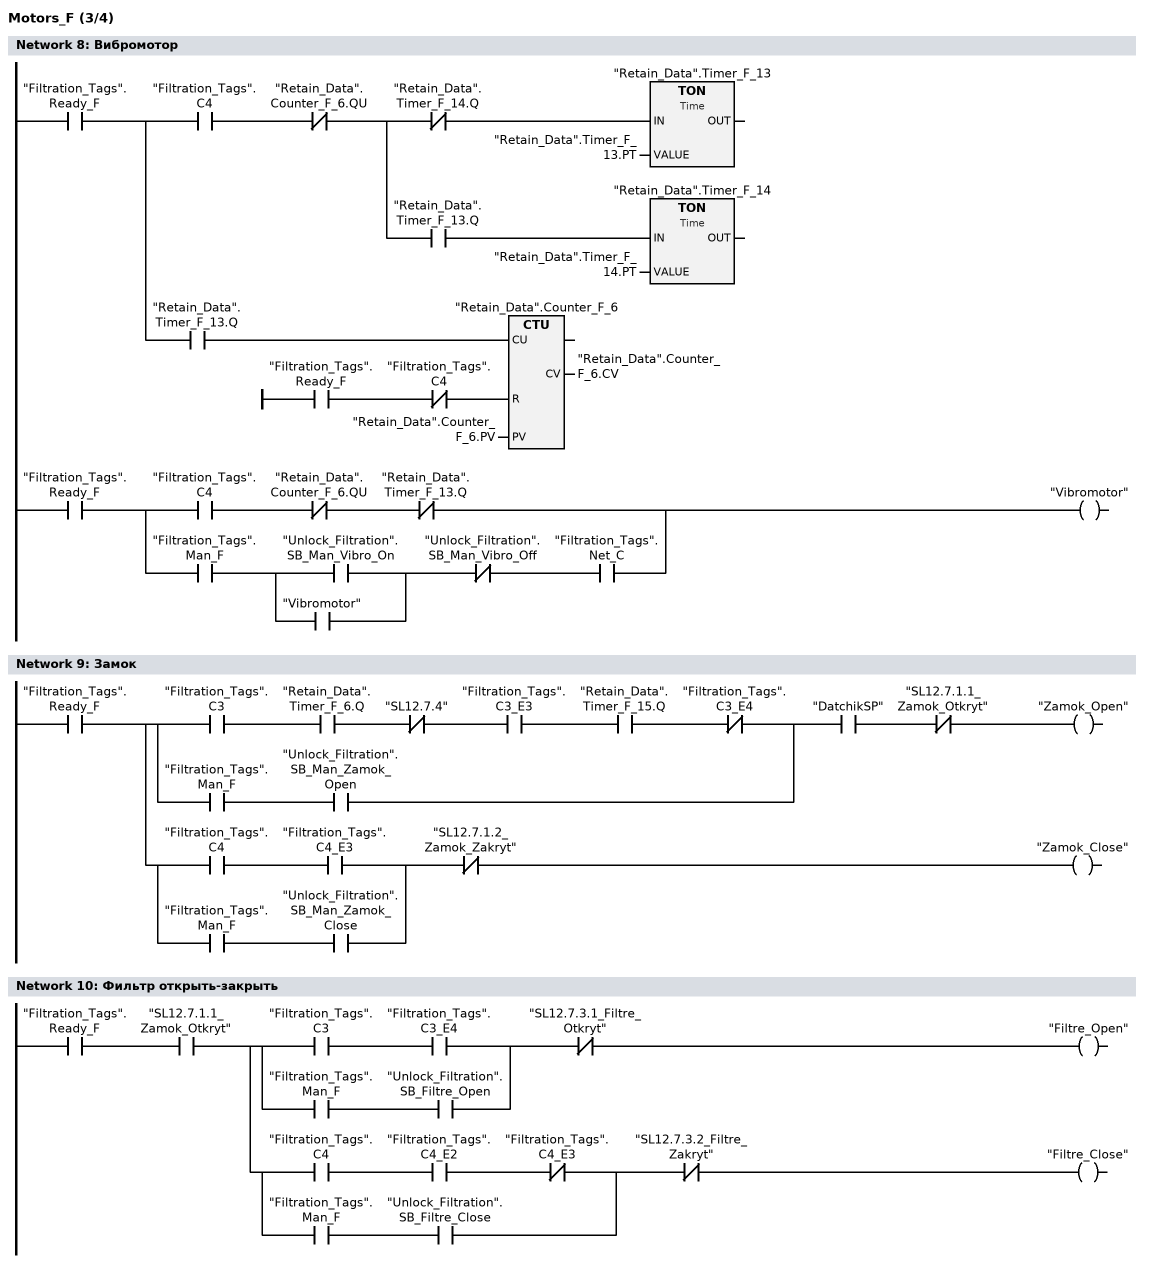
   #_w1 := "Filtration_Tags".Ready_F AND "Filtration_Tags".C4 AND NOT "Retain_Data".Counter_F_6.QU;
   "Retain_Data".Timer_F_13.TON(IN := #_w1 AND NOT "Retain_Data".Timer_F_14.Q, PT := "Retain_Data".Timer_F_13.PT);   // TON coil
   "Retain_Data".Timer_F_14.TON(IN := #_w1 AND "Retain_Data".Timer_F_13.Q, PT := "Retain_Data".Timer_F_14.PT);   // TON coil
   "Retain_Data".Counter_F_6.CTU(CU := "Filtration_Tags".Ready_F AND "Retain_Data".Timer_F_13.Q,
                           R := "Filtration_Tags".Ready_F AND NOT "Filtration_Tags".C4,
                           PV := "Retain_Data".Counter_F_6.PV,
                           CV => "Retain_Data".Counter_F_6.CV);
   "Vibromotor" := "Filtration_Tags".Ready_F AND (("Filtration_Tags".C4 AND NOT "Retain_Data".Counter_F_6.QU AND NOT "Retain_Data".Timer_F_13.Q) OR ("Filtration_Tags".Man_F AND ("Unlock_Filtration".SB_Man_Vibro_On OR "Vibromotor") AND NOT "Unlock_Filtration".SB_Man_Vibro_Off AND "Filtration_Tags".Net_C));
END_REGION

REGION Network 9: Замок
   RUNG wire#powerrail
      Contact( "Filtration_Tags".Ready_F )
      wire#w1
      Contact( "Filtration_Tags".C3 )
      Contact( "Retain_Data".Timer_F_6.Q )
      I_Contact( "SL12.7.4" )
      Contact( "Filtration_Tags".C3_E3 )
      Contact( "Retain_Data".Timer_F_15.Q )
      I_Contact( "Filtration_Tags".C3_E4 )
      wire#w2
      Contact( "DatchikSP" )
      I_Contact( "SL12.7.1.1_Zamok_Otkryt" )
      Coil( "Zamok_Open" )
   END_RUNG
   RUNG wire#w1
      Contact( "Filtration_Tags".Man_F )
      Contact( "Unlock_Filtration".SB_Man_Zamok_Open )
   END_RUNG wire#w2
   RUNG wire#w1
      Contact( "Filtration_Tags".C4 )
      Contact( "Filtration_Tags".C4_E3 )
      wire#w3
      I_Contact( "SL12.7.1.2_Zamok_Zakryt" )
      Coil( "Zamok_Close" )
   END_RUNG
   RUNG wire#w1
      Contact( "Filtration_Tags".Man_F )
      Contact( "Unlock_Filtration".SB_Man_Zamok_Close )
   END_RUNG wire#w3
   // the same network as SCL:
   "Zamok_Open" := "Filtration_Tags".Ready_F AND (("Filtration_Tags".C3 AND "Retain_Data".Timer_F_6.Q AND NOT "SL12.7.4" AND "Filtration_Tags".C3_E3 AND "Retain_Data".Timer_F_15.Q AND NOT "Filtration_Tags".C3_E4) OR ("Filtration_Tags".Man_F AND "Unlock_Filtration".SB_Man_Zamok_Open)) AND "DatchikSP" AND NOT "SL12.7.1.1_Zamok_Otkryt";
   "Zamok_Close" := "Filtration_Tags".Ready_F AND (("Filtration_Tags".C4 AND "Filtration_Tags".C4_E3) OR ("Filtration_Tags".Man_F AND "Unlock_Filtration".SB_Man_Zamok_Close)) AND NOT "SL12.7.1.2_Zamok_Zakryt";
END_REGION

REGION Network 10: Фильтр открыть-закрыть
   RUNG wire#powerrail
      Contact( "Filtration_Tags".Ready_F )
      Contact( "SL12.7.1.1_Zamok_Otkryt" )
      wire#w1
      Contact( "Filtration_Tags".C3 )
      Contact( "Filtration_Tags".C3_E4 )
      wire#w2
      I_Contact( "SL12.7.3.1_Filtre_Otkryt" )
      Coil( "Filtre_Open" )
   END_RUNG
   RUNG wire#w1
      Contact( "Filtration_Tags".Man_F )
      Contact( "Unlock_Filtration".SB_Filtre_Open )
   END_RUNG wire#w2
   RUNG wire#w1
      Contact( "Filtration_Tags".C4 )
      Contact( "Filtration_Tags".C4_E2 )
      I_Contact( "Filtration_Tags".C4_E3 )
      wire#w3
      I_Contact( "SL12.7.3.2_Filtre_Zakryt" )
      Coil( "Filtre_Close" )
   END_RUNG
   RUNG wire#w1
      Contact( "Filtration_Tags".Man_F )
      Contact( "Unlock_Filtration".SB_Filtre_Close )
   END_RUNG wire#w3
   // the same network as SCL:
   #_w1 := "Filtration_Tags".Ready_F AND "SL12.7.1.1_Zamok_Otkryt";
   "Filtre_Open" := #_w1 AND (("Filtration_Tags".C3 AND "Filtration_Tags".C3_E4) OR ("Filtration_Tags".Man_F AND "Unlock_Filtration".SB_Filtre_Open)) AND NOT "SL12.7.3.1_Filtre_Otkryt";
   "Filtre_Close" := #_w1 AND (("Filtration_Tags".C4 AND "Filtration_Tags".C4_E2 AND NOT "Filtration_Tags".C4_E3) OR ("Filtration_Tags".Man_F AND "Unlock_Filtration".SB_Filtre_Close)) AND NOT "SL12.7.3.2_Filtre_Zakryt";
END_REGION

REGION Network 11: Клапан K2.1
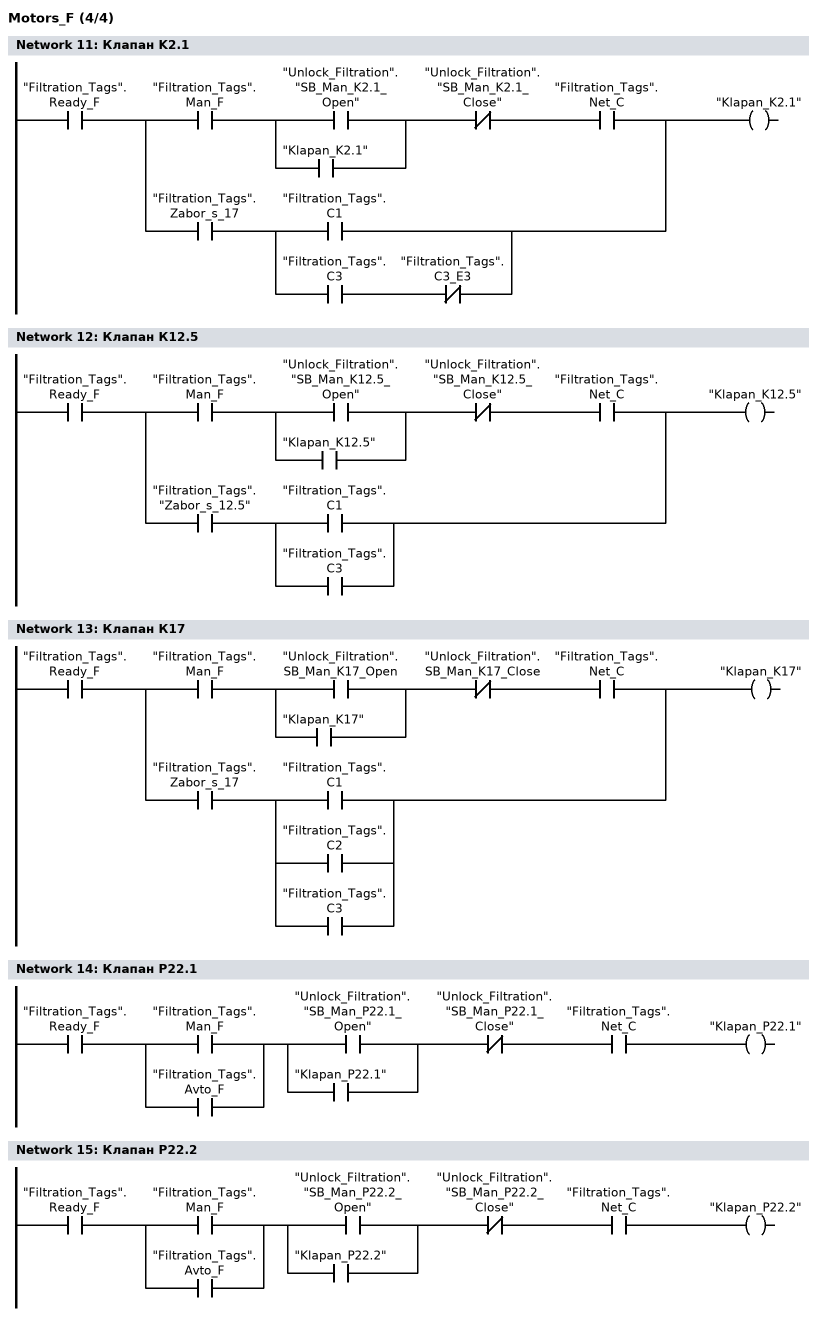
   RUNG wire#powerrail
      Contact( "Filtration_Tags".Ready_F )
      wire#w1
      Contact( "Filtration_Tags".Man_F )
      wire#w2
      Contact( "Unlock_Filtration"."SB_Man_K2.1_Open" )
      wire#w3
      I_Contact( "Unlock_Filtration"."SB_Man_K2.1_Close" )
      Contact( "Filtration_Tags".Net_C )
      wire#w4
      Coil( "Klapan_K2.1" )
   END_RUNG
   RUNG wire#w2
      Contact( "Klapan_K2.1" )
   END_RUNG wire#w3
   RUNG wire#w1
      Contact( "Filtration_Tags".Zabor_s_17 )
      wire#w5
      Contact( "Filtration_Tags".C1 )
   END_RUNG wire#w4
   RUNG wire#w5
      Contact( "Filtration_Tags".C3 )
      I_Contact( "Filtration_Tags".C3_E3 )
   END_RUNG wire#w4
   // the same network as SCL:
   "Klapan_K2.1" := "Filtration_Tags".Ready_F AND (("Filtration_Tags".Man_F AND ("Unlock_Filtration"."SB_Man_K2.1_Open" OR "Klapan_K2.1") AND NOT "Unlock_Filtration"."SB_Man_K2.1_Close" AND "Filtration_Tags".Net_C) OR ("Filtration_Tags".Zabor_s_17 AND ("Filtration_Tags".C1 OR ("Filtration_Tags".C3 AND NOT "Filtration_Tags".C3_E3))));
END_REGION

REGION Network 12: Клапан К12.5
   RUNG wire#powerrail
      Contact( "Filtration_Tags".Ready_F )
      wire#w1
      Contact( "Filtration_Tags".Man_F )
      wire#w2
      Contact( "Unlock_Filtration"."SB_Man_K12.5_Open" )
      wire#w3
      I_Contact( "Unlock_Filtration"."SB_Man_K12.5_Close" )
      Contact( "Filtration_Tags".Net_C )
      wire#w4
      Coil( "Klapan_K12.5" )
   END_RUNG
   RUNG wire#w2
      Contact( "Klapan_K12.5" )
   END_RUNG wire#w3
   RUNG wire#w1
      Contact( "Filtration_Tags"."Zabor_s_12.5" )
      wire#w5
      Contact( "Filtration_Tags".C1 )
   END_RUNG wire#w4
   RUNG wire#w5
      Contact( "Filtration_Tags".C3 )
   END_RUNG wire#w4
   // the same network as SCL:
   "Klapan_K12.5" := "Filtration_Tags".Ready_F AND (("Filtration_Tags".Man_F AND ("Unlock_Filtration"."SB_Man_K12.5_Open" OR "Klapan_K12.5") AND NOT "Unlock_Filtration"."SB_Man_K12.5_Close" AND "Filtration_Tags".Net_C) OR ("Filtration_Tags"."Zabor_s_12.5" AND ("Filtration_Tags".C1 OR "Filtration_Tags".C3)));
END_REGION

REGION Network 13: Клапан К17
   RUNG wire#powerrail
      Contact( "Filtration_Tags".Ready_F )
      wire#w1
      Contact( "Filtration_Tags".Man_F )
      wire#w2
      Contact( "Unlock_Filtration".SB_Man_K17_Open )
      wire#w3
      I_Contact( "Unlock_Filtration".SB_Man_K17_Close )
      Contact( "Filtration_Tags".Net_C )
      wire#w4
      Coil( "Klapan_K17" )
   END_RUNG
   RUNG wire#w2
      Contact( "Klapan_K17" )
   END_RUNG wire#w3
   RUNG wire#w1
      Contact( "Filtration_Tags".Zabor_s_17 )
      wire#w5
      Contact( "Filtration_Tags".C1 )
   END_RUNG wire#w4
   RUNG wire#w5
      Contact( "Filtration_Tags".C2 )
   END_RUNG wire#w4
   RUNG wire#w5
      Contact( "Filtration_Tags".C3 )
   END_RUNG wire#w4
   // the same network as SCL:
   "Klapan_K17" := "Filtration_Tags".Ready_F AND (("Filtration_Tags".Man_F AND ("Unlock_Filtration".SB_Man_K17_Open OR "Klapan_K17") AND NOT "Unlock_Filtration".SB_Man_K17_Close AND "Filtration_Tags".Net_C) OR ("Filtration_Tags".Zabor_s_17 AND ("Filtration_Tags".C1 OR "Filtration_Tags".C2 OR "Filtration_Tags".C3)));
END_REGION

REGION Network 14: Клапан P22.1
   RUNG wire#powerrail
      Contact( "Filtration_Tags".Ready_F )
      wire#w1
      Contact( "Filtration_Tags".Man_F )
      wire#w2
      Contact( "Unlock_Filtration"."SB_Man_P22.1_Open" )
      wire#w3
      I_Contact( "Unlock_Filtration"."SB_Man_P22.1_Close" )
      Contact( "Filtration_Tags".Net_C )
      Coil( "Klapan_P22.1" )
   END_RUNG
   RUNG wire#w1
      Contact( "Filtration_Tags".Avto_F )
   END_RUNG wire#w2
   RUNG wire#w2
      Contact( "Klapan_P22.1" )
   END_RUNG wire#w3
   // the same network as SCL:
   "Klapan_P22.1" := "Filtration_Tags".Ready_F AND ("Filtration_Tags".Man_F OR "Filtration_Tags".Avto_F) AND ("Unlock_Filtration"."SB_Man_P22.1_Open" OR "Klapan_P22.1") AND NOT "Unlock_Filtration"."SB_Man_P22.1_Close" AND "Filtration_Tags".Net_C;
END_REGION

REGION Network 15: Клапан P22.2
   RUNG wire#powerrail
      Contact( "Filtration_Tags".Ready_F )
      wire#w1
      Contact( "Filtration_Tags".Man_F )
      wire#w2
      Contact( "Unlock_Filtration"."SB_Man_P22.2_Open" )
      wire#w3
      I_Contact( "Unlock_Filtration"."SB_Man_P22.2_Close" )
      Contact( "Filtration_Tags".Net_C )
      Coil( "Klapan_P22.2" )
   END_RUNG
   RUNG wire#w1
      Contact( "Filtration_Tags".Avto_F )
   END_RUNG wire#w2
   RUNG wire#w2
      Contact( "Klapan_P22.2" )
   END_RUNG wire#w3
   // the same network as SCL:
   "Klapan_P22.2" := "Filtration_Tags".Ready_F AND ("Filtration_Tags".Man_F OR "Filtration_Tags".Avto_F) AND ("Unlock_Filtration"."SB_Man_P22.2_Open" OR "Klapan_P22.2") AND NOT "Unlock_Filtration"."SB_Man_P22.2_Close" AND "Filtration_Tags".Net_C;
END_REGION
END_FUNCTION_BLOCK

FUNCTION_BLOCK "Blokirovki"   // FB7, LAD
{ S7_Optimized_Access := 'TRUE' }
VERSION : 0.1
BEGIN

REGION Network 1: 7.5.1
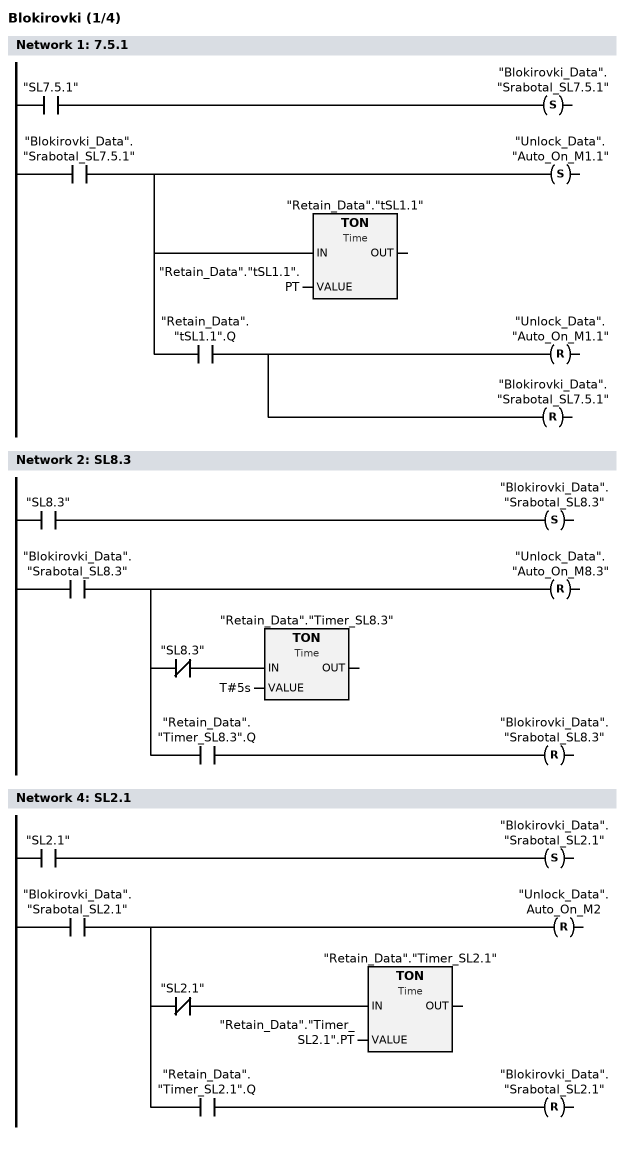
   IF "SL7.5.1" THEN "Blokirovki_Data"."Srabotal_SL7.5.1" := TRUE; END_IF;
   IF "Blokirovki_Data"."Srabotal_SL7.5.1" THEN "Unlock_Data"."Auto_On_M1.1" := TRUE; END_IF;
   "Retain_Data"."tSL1.1".TON(IN := "Blokirovki_Data"."Srabotal_SL7.5.1", PT := "Retain_Data"."tSL1.1".PT);   // TON coil
   IF "Blokirovki_Data"."Srabotal_SL7.5.1" AND "Retain_Data"."tSL1.1".Q THEN
       "Unlock_Data"."Auto_On_M1.1" := FALSE;
       "Blokirovki_Data"."Srabotal_SL7.5.1" := FALSE;
   END_IF;
END_REGION

REGION Network 2: SL8.3
   IF "SL8.3" THEN "Blokirovki_Data"."Srabotal_SL8.3" := TRUE; END_IF;
   IF "Blokirovki_Data"."Srabotal_SL8.3" THEN "Unlock_Data"."Auto_On_M8.3" := FALSE; END_IF;
   "Retain_Data"."Timer_SL8.3".TON(IN := "Blokirovki_Data"."Srabotal_SL8.3" AND NOT "SL8.3", PT := T#5s);   // TON coil
   IF "Blokirovki_Data"."Srabotal_SL8.3" AND "Retain_Data"."Timer_SL8.3".Q THEN
       "Blokirovki_Data"."Srabotal_SL8.3" := FALSE;
   END_IF;
END_REGION

REGION Network 4: SL2.1
   IF "SL2.1" THEN "Blokirovki_Data"."Srabotal_SL2.1" := TRUE; END_IF;
   IF "Blokirovki_Data"."Srabotal_SL2.1" THEN "Unlock_Data".Auto_On_M2 := FALSE; END_IF;
   "Retain_Data"."Timer_SL2.1".TON(IN := "Blokirovki_Data"."Srabotal_SL2.1" AND NOT "SL2.1", PT := "Retain_Data"."Timer_SL2.1".PT);   // TON coil
   IF "Blokirovki_Data"."Srabotal_SL2.1" AND "Retain_Data"."Timer_SL2.1".Q THEN
       "Blokirovki_Data"."Srabotal_SL2.1" := FALSE;
   END_IF;
END_REGION

REGION Network 5: SL5.1
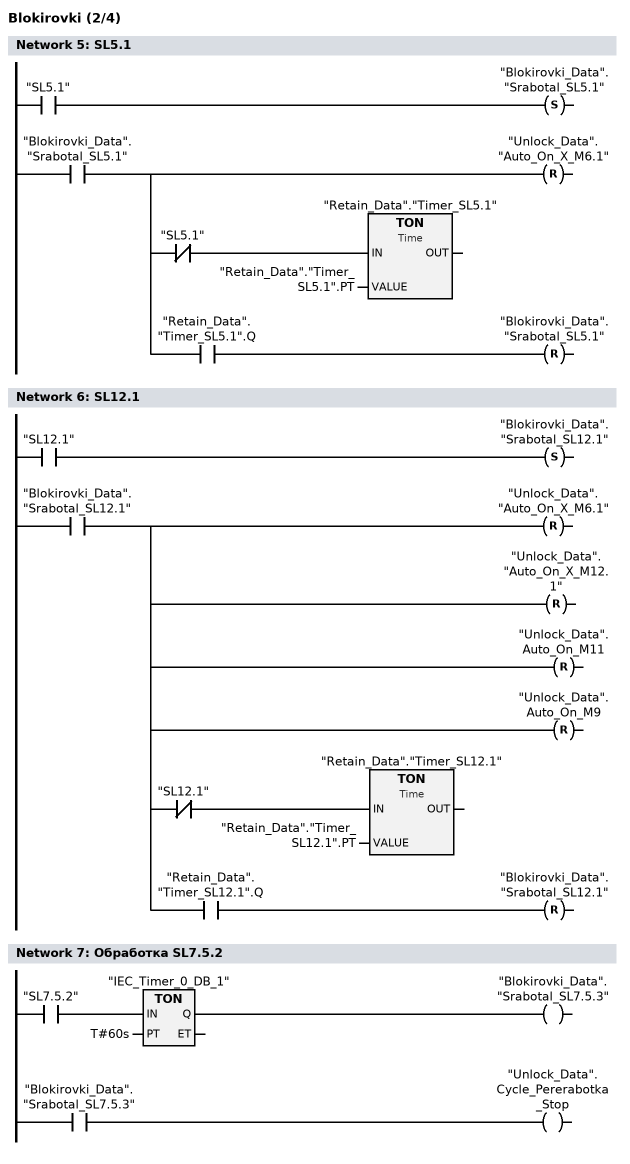
   IF "SL5.1" THEN "Blokirovki_Data"."Srabotal_SL5.1" := TRUE; END_IF;
   IF "Blokirovki_Data"."Srabotal_SL5.1" THEN "Unlock_Data"."Auto_On_X_M6.1" := FALSE; END_IF;
   "Retain_Data"."Timer_SL5.1".TON(IN := "Blokirovki_Data"."Srabotal_SL5.1" AND NOT "SL5.1", PT := "Retain_Data"."Timer_SL5.1".PT);   // TON coil
   IF "Blokirovki_Data"."Srabotal_SL5.1" AND "Retain_Data"."Timer_SL5.1".Q THEN
       "Blokirovki_Data"."Srabotal_SL5.1" := FALSE;
   END_IF;
END_REGION

REGION Network 6: SL12.1
   IF "SL12.1" THEN "Blokirovki_Data"."Srabotal_SL12.1" := TRUE; END_IF;
   IF "Blokirovki_Data"."Srabotal_SL12.1" THEN
       "Unlock_Data"."Auto_On_X_M6.1" := FALSE;
       "Unlock_Data"."Auto_On_X_M12.1" := FALSE;
       "Unlock_Data".Auto_On_M11 := FALSE;
       "Unlock_Data".Auto_On_M9 := FALSE;
   END_IF;
   "Retain_Data"."Timer_SL12.1".TON(IN := "Blokirovki_Data"."Srabotal_SL12.1" AND NOT "SL12.1", PT := "Retain_Data"."Timer_SL12.1".PT);   // TON coil
   IF "Blokirovki_Data"."Srabotal_SL12.1" AND "Retain_Data"."Timer_SL12.1".Q THEN
       "Blokirovki_Data"."Srabotal_SL12.1" := FALSE;
   END_IF;
END_REGION

REGION Network 7: Обработка SL7.5.2
   "IEC_Timer_0_DB_1".TON(IN := "SL7.5.2", PT := T#60s);
   "Blokirovki_Data"."Srabotal_SL7.5.3" := "IEC_Timer_0_DB_1".Q;
   "Unlock_Data".Cycle_Pererabotka_Stop := "Blokirovki_Data"."Srabotal_SL7.5.3";
END_REGION

REGION Network 8: SL9.1
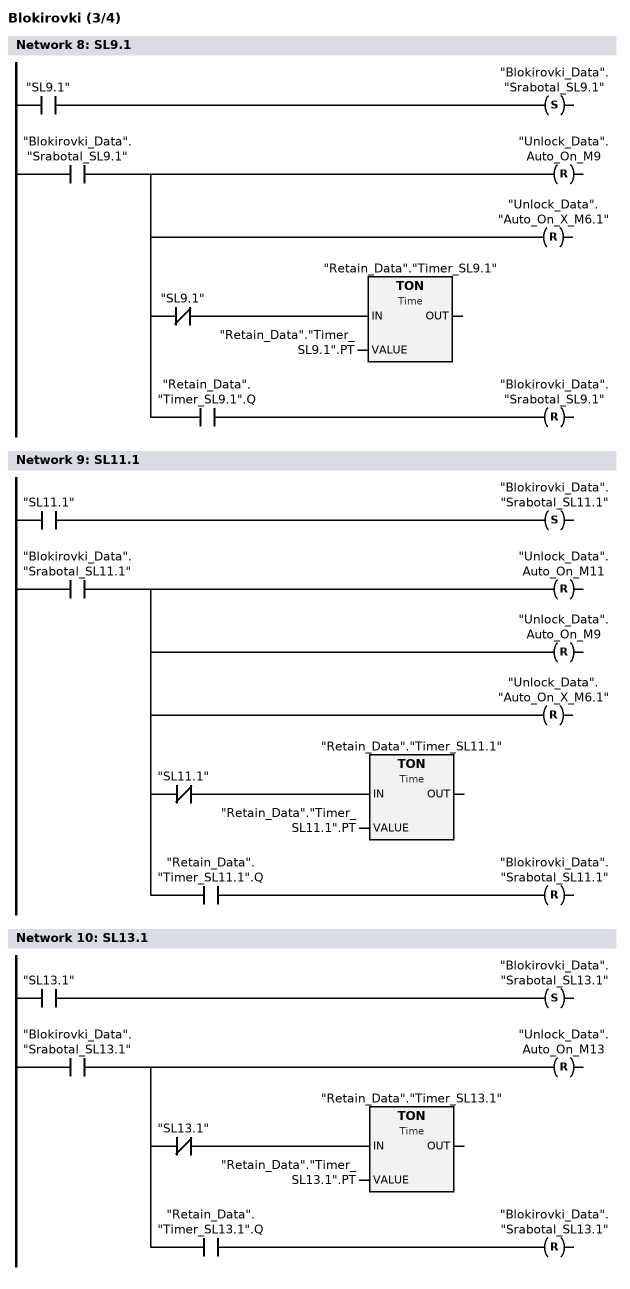
   IF "SL9.1" THEN "Blokirovki_Data"."Srabotal_SL9.1" := TRUE; END_IF;
   IF "Blokirovki_Data"."Srabotal_SL9.1" THEN
       "Unlock_Data".Auto_On_M9 := FALSE;
       "Unlock_Data"."Auto_On_X_M6.1" := FALSE;
   END_IF;
   "Retain_Data"."Timer_SL9.1".TON(IN := "Blokirovki_Data"."Srabotal_SL9.1" AND NOT "SL9.1", PT := "Retain_Data"."Timer_SL9.1".PT);   // TON coil
   IF "Blokirovki_Data"."Srabotal_SL9.1" AND "Retain_Data"."Timer_SL9.1".Q THEN
       "Blokirovki_Data"."Srabotal_SL9.1" := FALSE;
   END_IF;
END_REGION

REGION Network 9: SL11.1
   IF "SL11.1" THEN "Blokirovki_Data"."Srabotal_SL11.1" := TRUE; END_IF;
   IF "Blokirovki_Data"."Srabotal_SL11.1" THEN
       "Unlock_Data".Auto_On_M11 := FALSE;
       "Unlock_Data".Auto_On_M9 := FALSE;
       "Unlock_Data"."Auto_On_X_M6.1" := FALSE;
   END_IF;
   "Retain_Data"."Timer_SL11.1".TON(IN := "Blokirovki_Data"."Srabotal_SL11.1" AND NOT "SL11.1", PT := "Retain_Data"."Timer_SL11.1".PT);   // TON coil
   IF "Blokirovki_Data"."Srabotal_SL11.1" AND "Retain_Data"."Timer_SL11.1".Q THEN
       "Blokirovki_Data"."Srabotal_SL11.1" := FALSE;
   END_IF;
END_REGION

REGION Network 10: SL13.1
   IF "SL13.1" THEN "Blokirovki_Data"."Srabotal_SL13.1" := TRUE; END_IF;
   IF "Blokirovki_Data"."Srabotal_SL13.1" THEN "Unlock_Data".Auto_On_M13 := FALSE; END_IF;
   "Retain_Data"."Timer_SL13.1".TON(IN := "Blokirovki_Data"."Srabotal_SL13.1" AND NOT "SL13.1", PT := "Retain_Data"."Timer_SL13.1".PT);   // TON coil
   IF "Blokirovki_Data"."Srabotal_SL13.1" AND "Retain_Data"."Timer_SL13.1".Q THEN
       "Blokirovki_Data"."Srabotal_SL13.1" := FALSE;
   END_IF;
END_REGION

REGION Network 11: Работа насоса М15
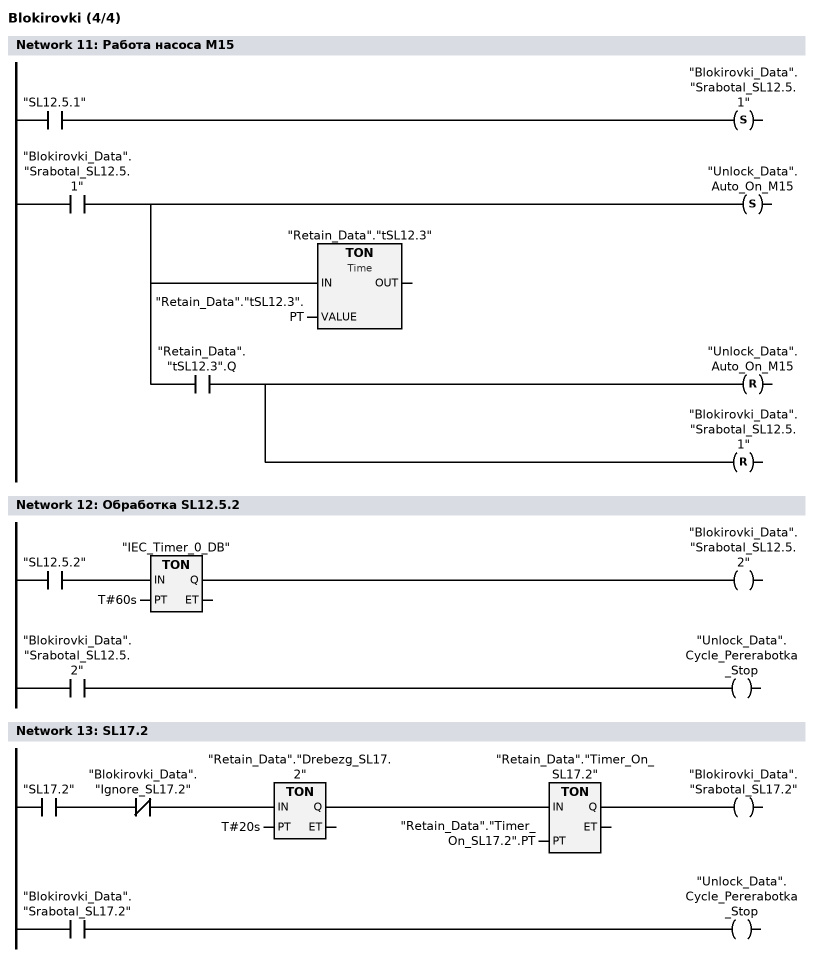
   IF "SL12.5.1" THEN "Blokirovki_Data"."Srabotal_SL12.5.1" := TRUE; END_IF;
   IF "Blokirovki_Data"."Srabotal_SL12.5.1" THEN "Unlock_Data".Auto_On_M15 := TRUE; END_IF;
   "Retain_Data"."tSL12.3".TON(IN := "Blokirovki_Data"."Srabotal_SL12.5.1", PT := "Retain_Data"."tSL12.3".PT);   // TON coil
   IF "Blokirovki_Data"."Srabotal_SL12.5.1" AND "Retain_Data"."tSL12.3".Q THEN
       "Unlock_Data".Auto_On_M15 := FALSE;
       "Blokirovki_Data"."Srabotal_SL12.5.1" := FALSE;
   END_IF;
END_REGION

REGION Network 12: Обработка SL12.5.2
   "IEC_Timer_0_DB".TON(IN := "SL12.5.2", PT := T#60s);
   "Blokirovki_Data"."Srabotal_SL12.5.2" := "IEC_Timer_0_DB".Q;
   "Unlock_Data".Cycle_Pererabotka_Stop := "Blokirovki_Data"."Srabotal_SL12.5.2";
END_REGION

REGION Network 13: SL17.2
   "Retain_Data"."Drebezg_SL17.2".TON(IN := "SL17.2" AND NOT "Blokirovki_Data"."Ignore_SL17.2", PT := T#20s);
   "Retain_Data"."Timer_On_SL17.2".TON(IN := "Retain_Data"."Drebezg_SL17.2".Q,
                           PT := "Retain_Data"."Timer_On_SL17.2".PT);
   "Blokirovki_Data"."Srabotal_SL17.2" := "Retain_Data"."Timer_On_SL17.2".Q;
   "Unlock_Data".Cycle_Pererabotka_Stop := "Blokirovki_Data"."Srabotal_SL17.2";
END_REGION

REGION Network 14: Обработка SL22.1
END_REGION

REGION Network 15: Обработка SL22.2
END_REGION
END_FUNCTION_BLOCK

FUNCTION_BLOCK "Lamp_Sound"   // FB8, LAD
{ S7_Optimized_Access := 'TRUE' }
VERSION : 0.1
BEGIN

REGION Network 1
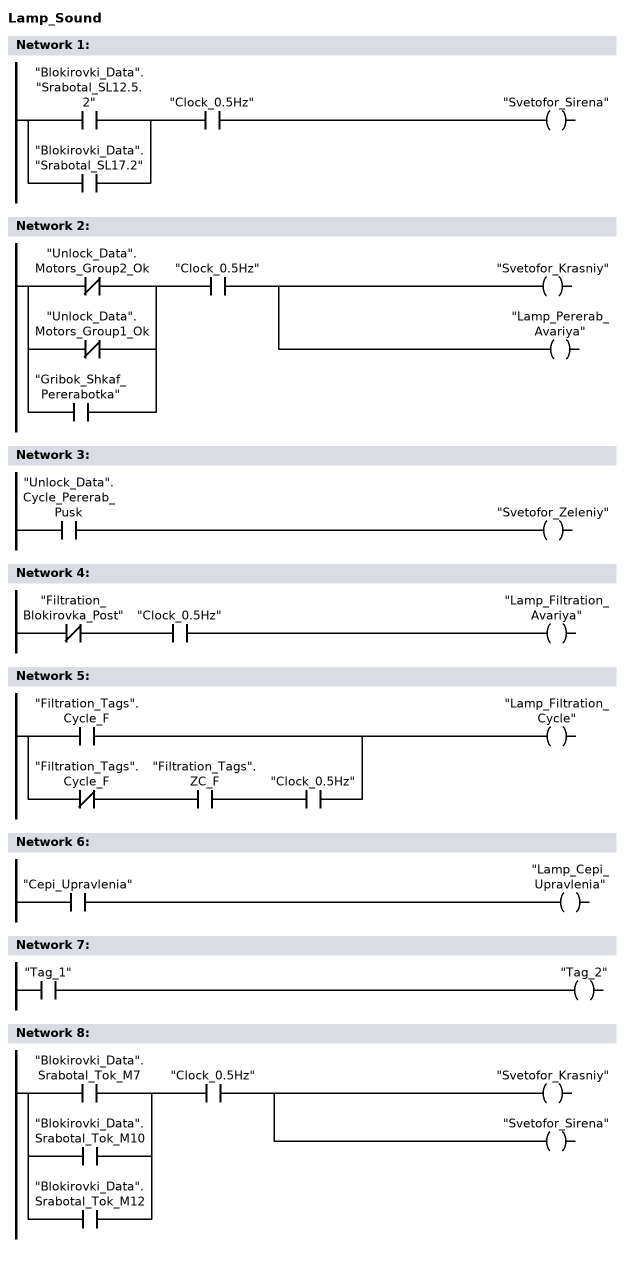
   RUNG wire#powerrail
      Contact( "Blokirovki_Data"."Srabotal_SL12.5.2" )
      wire#w1
      Contact( "Clock_0.5Hz" )
      Coil( "Svetofor_Sirena" )
   END_RUNG
   RUNG wire#powerrail
      Contact( "Blokirovki_Data"."Srabotal_SL17.2" )
   END_RUNG wire#w1
   // the same network as SCL:
   "Svetofor_Sirena" := ("Blokirovki_Data"."Srabotal_SL12.5.2" OR "Blokirovki_Data"."Srabotal_SL17.2") AND "Clock_0.5Hz";
END_REGION

REGION Network 2
   RUNG wire#powerrail
      I_Contact( "Unlock_Data".Motors_Group2_Ok )
      wire#w1
      Contact( "Clock_0.5Hz" )
      wire#w2
      Coil( "Svetofor_Krasniy" )
   END_RUNG
   RUNG wire#powerrail
      I_Contact( "Unlock_Data".Motors_Group1_Ok )
   END_RUNG wire#w1
   RUNG wire#powerrail
      Contact( "Gribok_Shkaf_Pererabotka" )
   END_RUNG wire#w1
   RUNG wire#w2
      Coil( "Lamp_Pererab_Avariya" )
   END_RUNG
   // the same network as SCL:
   "Svetofor_Krasniy" := (NOT "Unlock_Data".Motors_Group2_Ok OR NOT "Unlock_Data".Motors_Group1_Ok OR "Gribok_Shkaf_Pererabotka") AND "Clock_0.5Hz";
   "Lamp_Pererab_Avariya" := "Svetofor_Krasniy";
END_REGION

REGION Network 3
   RUNG wire#powerrail
      Contact( "Unlock_Data".Cycle_Pererab_Pusk )
      Coil( "Svetofor_Zeleniy" )
   END_RUNG
   // the same network as SCL:
   "Svetofor_Zeleniy" := "Unlock_Data".Cycle_Pererab_Pusk;
END_REGION

REGION Network 4
   RUNG wire#powerrail
      I_Contact( "Filtration_Blokirovka_Post" )
      Contact( "Clock_0.5Hz" )
      Coil( "Lamp_Filtration_Avariya" )
   END_RUNG
   // the same network as SCL:
   "Lamp_Filtration_Avariya" := NOT "Filtration_Blokirovka_Post" AND "Clock_0.5Hz";
END_REGION

REGION Network 5
   RUNG wire#powerrail
      Contact( "Filtration_Tags".Cycle_F )
      wire#w1
      Coil( "Lamp_Filtration_Cycle" )
   END_RUNG
   RUNG wire#powerrail
      I_Contact( "Filtration_Tags".Cycle_F )
      Contact( "Filtration_Tags".ZC_F )
      Contact( "Clock_0.5Hz" )
   END_RUNG wire#w1
   // the same network as SCL:
   "Lamp_Filtration_Cycle" := "Filtration_Tags".Cycle_F OR (NOT "Filtration_Tags".Cycle_F AND "Filtration_Tags".ZC_F AND "Clock_0.5Hz");
END_REGION

REGION Network 6
   RUNG wire#powerrail
      Contact( "Cepi_Upravlenia" )
      Coil( "Lamp_Cepi_Upravlenia" )
   END_RUNG
   // the same network as SCL:
   "Lamp_Cepi_Upravlenia" := "Cepi_Upravlenia";
END_REGION

REGION Network 7
   RUNG wire#powerrail
      Contact( "Tag_1" )
      Coil( "Tag_2" )
   END_RUNG
   // the same network as SCL:
   "Tag_2" := "Tag_1";
END_REGION

REGION Network 8
   RUNG wire#powerrail
      Contact( "Blokirovki_Data".Srabotal_Tok_M7 )
      wire#w1
      Contact( "Clock_0.5Hz" )
      wire#w2
      Coil( "Svetofor_Krasniy" )
   END_RUNG
   RUNG wire#powerrail
      Contact( "Blokirovki_Data".Srabotal_Tok_M10 )
   END_RUNG wire#w1
   RUNG wire#powerrail
      Contact( "Blokirovki_Data".Srabotal_Tok_M12 )
   END_RUNG wire#w1
   RUNG wire#w2
      Coil( "Svetofor_Sirena" )
   END_RUNG
   // the same network as SCL:
   "Svetofor_Krasniy" := ("Blokirovki_Data".Srabotal_Tok_M7 OR "Blokirovki_Data".Srabotal_Tok_M10 OR "Blokirovki_Data".Srabotal_Tok_M12) AND "Clock_0.5Hz";
   "Svetofor_Sirena" := "Svetofor_Krasniy";
END_REGION
END_FUNCTION_BLOCK

FUNCTION_BLOCK "Temper_Tok"   // FB9, LAD
{ S7_Optimized_Access := 'TRUE' }
VERSION : 0.1
   VAR_TEMP   // added for the SCL form of the ladder/FBD networks
      _w1 : Bool;
   END_VAR
BEGIN

REGION Network 1
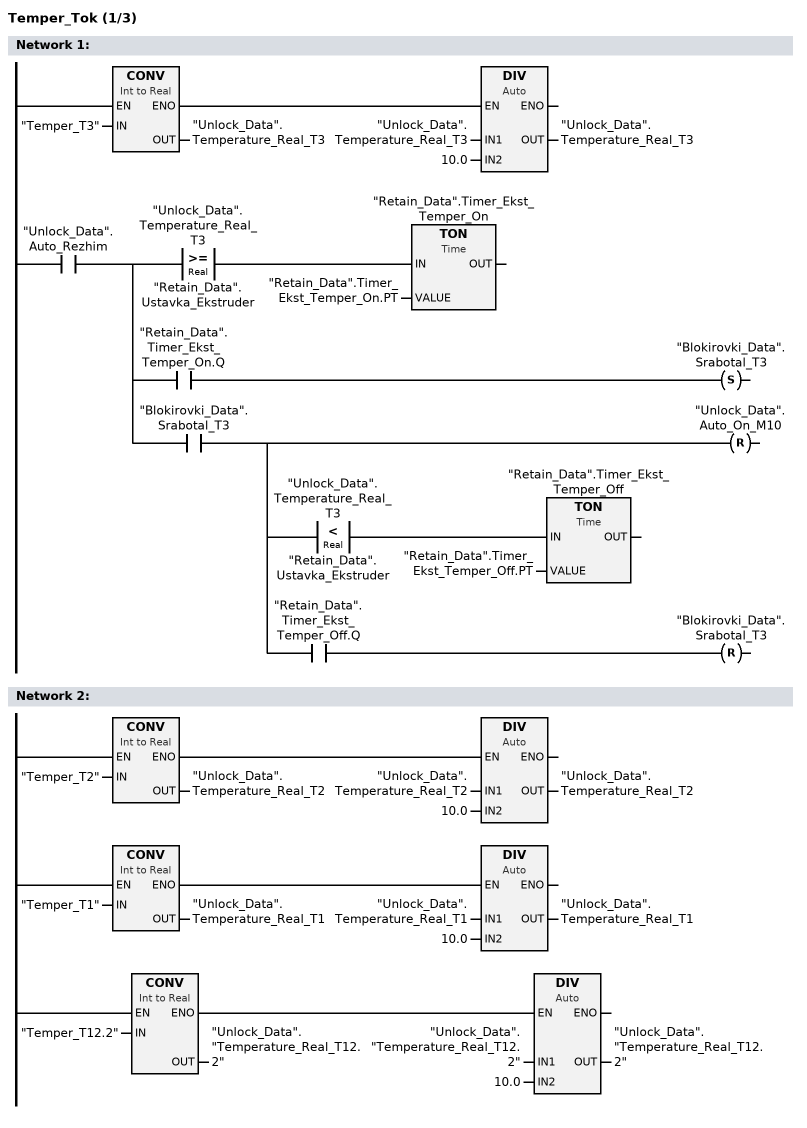
   "Unlock_Data".Temperature_Real_T3 := INT_TO_REAL("Temper_T3");
   "Unlock_Data".Temperature_Real_T3 := "Unlock_Data".Temperature_Real_T3 / 10.0;
   "Retain_Data".Timer_Ekst_Temper_On.TON(IN := "Unlock_Data".Auto_Rezhim AND ("Unlock_Data".Temperature_Real_T3 >= "Retain_Data".Ustavka_Ekstruder), PT := "Retain_Data".Timer_Ekst_Temper_On.PT);   // TON coil
   IF "Unlock_Data".Auto_Rezhim AND "Retain_Data".Timer_Ekst_Temper_On.Q THEN
       "Blokirovki_Data".Srabotal_T3 := TRUE;
   END_IF;
   #_w1 := "Unlock_Data".Auto_Rezhim AND "Blokirovki_Data".Srabotal_T3;
   IF #_w1 THEN "Unlock_Data".Auto_On_M10 := FALSE; END_IF;
   "Retain_Data".Timer_Ekst_Temper_Off.TON(IN := #_w1 AND ("Unlock_Data".Temperature_Real_T3 < "Retain_Data".Ustavka_Ekstruder), PT := "Retain_Data".Timer_Ekst_Temper_Off.PT);   // TON coil
   IF #_w1 AND "Retain_Data".Timer_Ekst_Temper_Off.Q THEN "Blokirovki_Data".Srabotal_T3 := FALSE; END_IF;
END_REGION

REGION Network 2
   RUNG wire#powerrail
      { S7_Templates := "[SrcType := Int, DestType := Real]" } Convert(in := "Temper_T2", out => "Unlock_Data".Temperature_Real_T2)
      Div(in1 := "Unlock_Data".Temperature_Real_T2, in2 := 10.0, out => "Unlock_Data".Temperature_Real_T2)
   END_RUNG
   RUNG wire#powerrail
      { S7_Templates := "[SrcType := Int, DestType := Real]" } Convert(in := "Temper_T1", out => "Unlock_Data".Temperature_Real_T1)
      Div(in1 := "Unlock_Data".Temperature_Real_T1, in2 := 10.0, out => "Unlock_Data".Temperature_Real_T1)
   END_RUNG
   RUNG wire#powerrail
      { S7_Templates := "[SrcType := Int, DestType := Real]" } Convert(in := "Temper_T12.2", out => "Unlock_Data"."Temperature_Real_T12.2")
      Div(in1 := "Unlock_Data"."Temperature_Real_T12.2", in2 := 10.0, out => "Unlock_Data"."Temperature_Real_T12.2")
   END_RUNG
   // the same network as SCL:
   "Unlock_Data".Temperature_Real_T2 := INT_TO_REAL("Temper_T2");
   "Unlock_Data".Temperature_Real_T2 := "Unlock_Data".Temperature_Real_T2 / 10.0;
   "Unlock_Data".Temperature_Real_T1 := INT_TO_REAL("Temper_T1");
   "Unlock_Data".Temperature_Real_T1 := "Unlock_Data".Temperature_Real_T1 / 10.0;
   "Unlock_Data"."Temperature_Real_T12.2" := INT_TO_REAL("Temper_T12.2");
   "Unlock_Data"."Temperature_Real_T12.2" := "Unlock_Data"."Temperature_Real_T12.2" / 10.0;
END_REGION

REGION Network 3
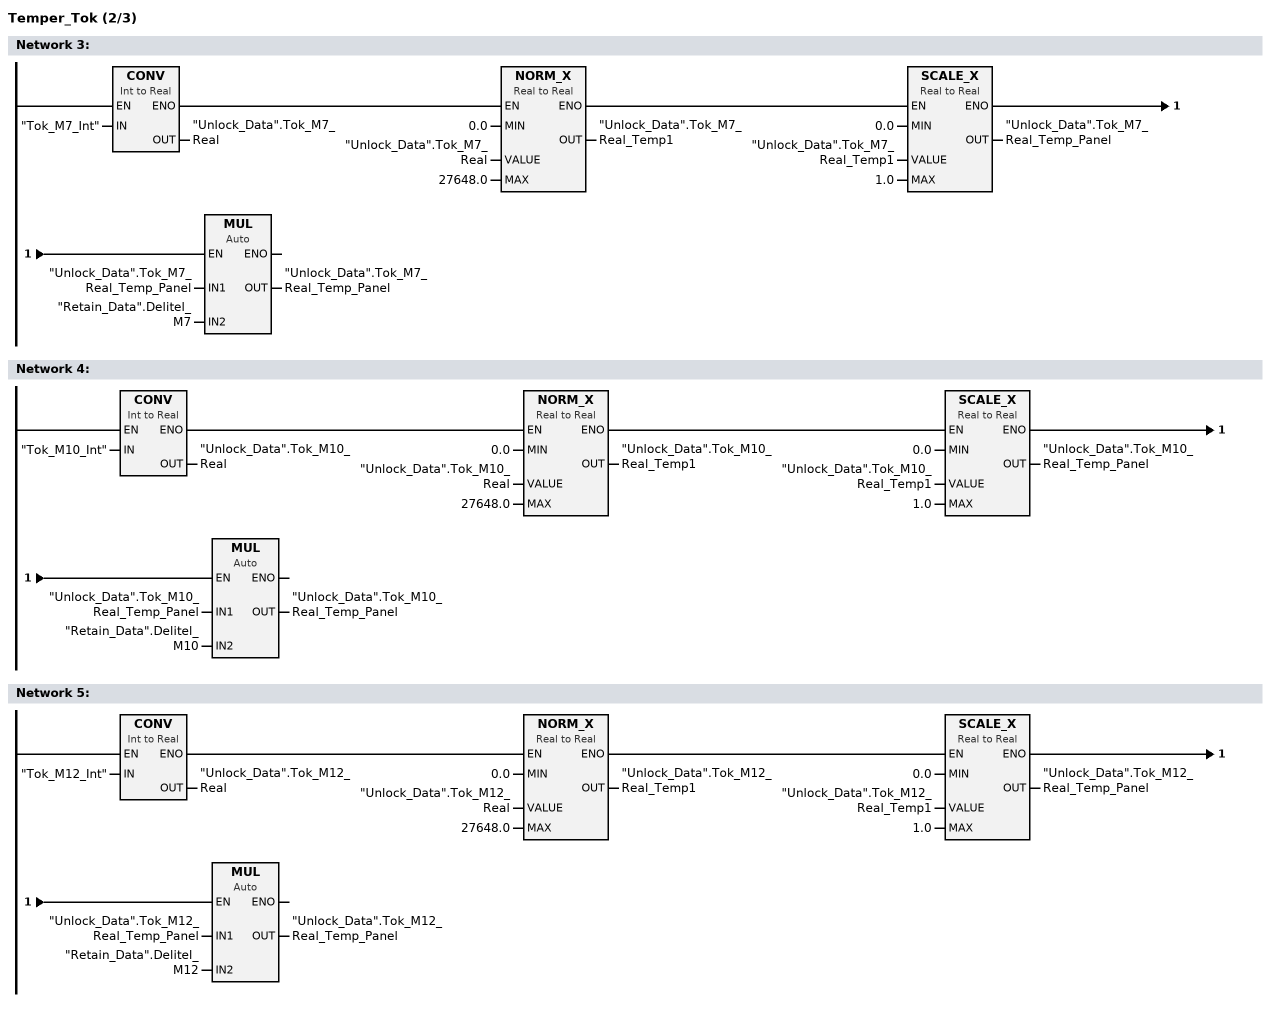
   RUNG wire#powerrail
      { S7_Templates := "[SrcType := Int, DestType := Real]" } Convert(in := "Tok_M7_Int", out => "Unlock_Data".Tok_M7_Real)
      { S7_Templates := "[SrcType := Real, DestType := Real]" } Normalize(min := 0.0, value := "Unlock_Data".Tok_M7_Real, max := 27648.0, out => "Unlock_Data".Tok_M7_Real_Temp1)
      { S7_Templates := "[SrcType := Real, DestType := Real]" } Scale(min := 0.0, value := "Unlock_Data".Tok_M7_Real_Temp1, max := 1.0, out => "Unlock_Data".Tok_M7_Real_Temp_Panel)
      Mul(in1 := "Unlock_Data".Tok_M7_Real_Temp_Panel, in2 := "Retain_Data".Delitel_M7, out => "Unlock_Data".Tok_M7_Real_Temp_Panel)
   END_RUNG
   // the same network as SCL:
   "Unlock_Data".Tok_M7_Real := INT_TO_REAL("Tok_M7_Int");
   "Unlock_Data".Tok_M7_Real_Temp1 := NORM_X(MIN := 0.0, VALUE := "Unlock_Data".Tok_M7_Real, MAX := 27648.0);
   "Unlock_Data".Tok_M7_Real_Temp_Panel := SCALE_X(MIN := 0.0, VALUE := "Unlock_Data".Tok_M7_Real_Temp1, MAX := 1.0);
   "Unlock_Data".Tok_M7_Real_Temp_Panel := "Unlock_Data".Tok_M7_Real_Temp_Panel * "Retain_Data".Delitel_M7;
END_REGION

REGION Network 4
   RUNG wire#powerrail
      { S7_Templates := "[SrcType := Int, DestType := Real]" } Convert(in := "Tok_M10_Int", out => "Unlock_Data".Tok_M10_Real)
      { S7_Templates := "[SrcType := Real, DestType := Real]" } Normalize(min := 0.0, value := "Unlock_Data".Tok_M10_Real, max := 27648.0, out => "Unlock_Data".Tok_M10_Real_Temp1)
      { S7_Templates := "[SrcType := Real, DestType := Real]" } Scale(min := 0.0, value := "Unlock_Data".Tok_M10_Real_Temp1, max := 1.0, out => "Unlock_Data".Tok_M10_Real_Temp_Panel)
      Mul(in1 := "Unlock_Data".Tok_M10_Real_Temp_Panel, in2 := "Retain_Data".Delitel_M10, out => "Unlock_Data".Tok_M10_Real_Temp_Panel)
   END_RUNG
   // the same network as SCL:
   "Unlock_Data".Tok_M10_Real := INT_TO_REAL("Tok_M10_Int");
   "Unlock_Data".Tok_M10_Real_Temp1 := NORM_X(MIN := 0.0, VALUE := "Unlock_Data".Tok_M10_Real, MAX := 27648.0);
   "Unlock_Data".Tok_M10_Real_Temp_Panel := SCALE_X(MIN := 0.0, VALUE := "Unlock_Data".Tok_M10_Real_Temp1, MAX := 1.0);
   "Unlock_Data".Tok_M10_Real_Temp_Panel := "Unlock_Data".Tok_M10_Real_Temp_Panel * "Retain_Data".Delitel_M10;
END_REGION

REGION Network 5
   RUNG wire#powerrail
      { S7_Templates := "[SrcType := Int, DestType := Real]" } Convert(in := "Tok_M12_Int", out => "Unlock_Data".Tok_M12_Real)
      { S7_Templates := "[SrcType := Real, DestType := Real]" } Normalize(min := 0.0, value := "Unlock_Data".Tok_M12_Real, max := 27648.0, out => "Unlock_Data".Tok_M12_Real_Temp1)
      { S7_Templates := "[SrcType := Real, DestType := Real]" } Scale(min := 0.0, value := "Unlock_Data".Tok_M12_Real_Temp1, max := 1.0, out => "Unlock_Data".Tok_M12_Real_Temp_Panel)
      Mul(in1 := "Unlock_Data".Tok_M12_Real_Temp_Panel, in2 := "Retain_Data".Delitel_M12, out => "Unlock_Data".Tok_M12_Real_Temp_Panel)
   END_RUNG
   // the same network as SCL:
   "Unlock_Data".Tok_M12_Real := INT_TO_REAL("Tok_M12_Int");
   "Unlock_Data".Tok_M12_Real_Temp1 := NORM_X(MIN := 0.0, VALUE := "Unlock_Data".Tok_M12_Real, MAX := 27648.0);
   "Unlock_Data".Tok_M12_Real_Temp_Panel := SCALE_X(MIN := 0.0, VALUE := "Unlock_Data".Tok_M12_Real_Temp1, MAX := 1.0);
   "Unlock_Data".Tok_M12_Real_Temp_Panel := "Unlock_Data".Tok_M12_Real_Temp_Panel * "Retain_Data".Delitel_M12;
END_REGION

REGION Network 6: Превышение тока m7
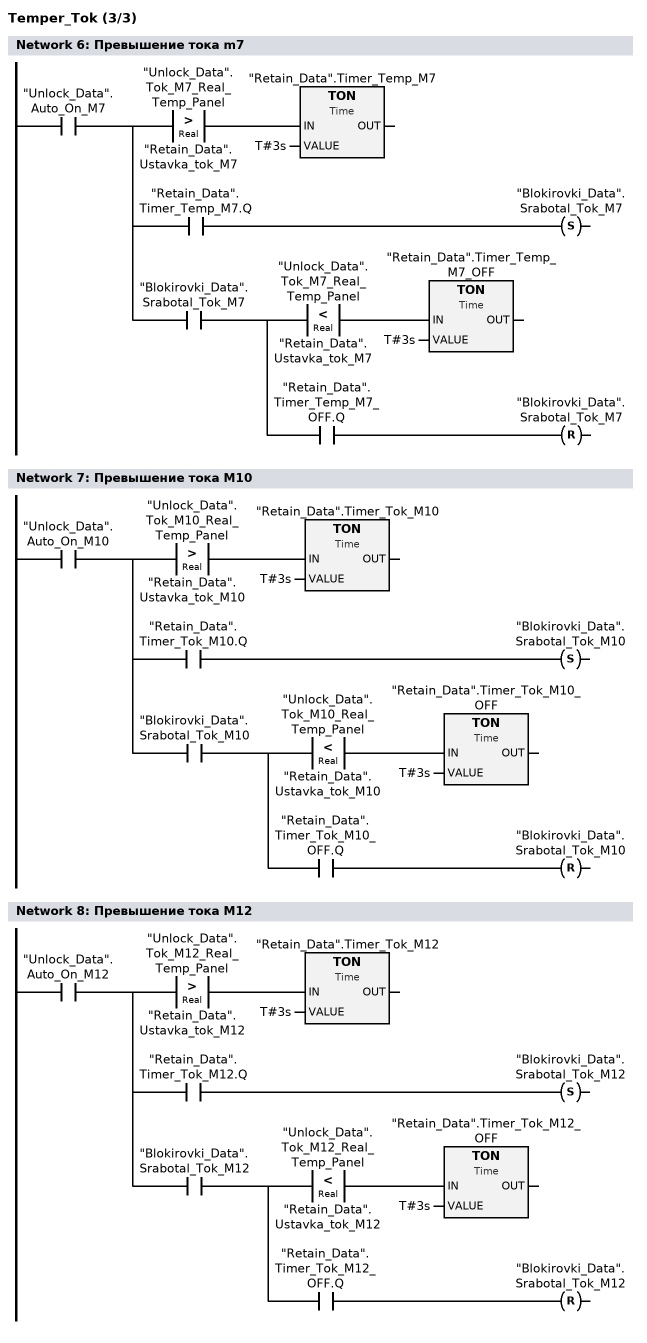
   "Retain_Data".Timer_Temp_M7.TON(IN := "Unlock_Data".Auto_On_M7 AND ("Unlock_Data".Tok_M7_Real_Temp_Panel > "Retain_Data".Ustavka_tok_M7), PT := T#3s);   // TON coil
   IF "Unlock_Data".Auto_On_M7 AND "Retain_Data".Timer_Temp_M7.Q THEN
       "Blokirovki_Data".Srabotal_Tok_M7 := TRUE;
   END_IF;
   #_w1 := "Unlock_Data".Auto_On_M7 AND "Blokirovki_Data".Srabotal_Tok_M7;
   "Retain_Data".Timer_Temp_M7_OFF.TON(IN := #_w1 AND ("Unlock_Data".Tok_M7_Real_Temp_Panel < "Retain_Data".Ustavka_tok_M7), PT := T#3s);   // TON coil
   IF #_w1 AND "Retain_Data".Timer_Temp_M7_OFF.Q THEN "Blokirovki_Data".Srabotal_Tok_M7 := FALSE; END_IF;
END_REGION

REGION Network 7: Превышение тока М10
   "Retain_Data".Timer_Tok_M10.TON(IN := "Unlock_Data".Auto_On_M10 AND ("Unlock_Data".Tok_M10_Real_Temp_Panel > "Retain_Data".Ustavka_tok_M10), PT := T#3s);   // TON coil
   IF "Unlock_Data".Auto_On_M10 AND "Retain_Data".Timer_Tok_M10.Q THEN
       "Blokirovki_Data".Srabotal_Tok_M10 := TRUE;
   END_IF;
   #_w1 := "Unlock_Data".Auto_On_M10 AND "Blokirovki_Data".Srabotal_Tok_M10;
   "Retain_Data".Timer_Tok_M10_OFF.TON(IN := #_w1 AND ("Unlock_Data".Tok_M10_Real_Temp_Panel < "Retain_Data".Ustavka_tok_M10), PT := T#3s);   // TON coil
   IF #_w1 AND "Retain_Data".Timer_Tok_M10_OFF.Q THEN "Blokirovki_Data".Srabotal_Tok_M10 := FALSE; END_IF;
END_REGION

REGION Network 8: Превышение тока М12
   "Retain_Data".Timer_Tok_M12.TON(IN := "Unlock_Data".Auto_On_M12 AND ("Unlock_Data".Tok_M12_Real_Temp_Panel > "Retain_Data".Ustavka_tok_M12), PT := T#3s);   // TON coil
   IF "Unlock_Data".Auto_On_M12 AND "Retain_Data".Timer_Tok_M12.Q THEN
       "Blokirovki_Data".Srabotal_Tok_M12 := TRUE;
   END_IF;
   #_w1 := "Unlock_Data".Auto_On_M12 AND "Blokirovki_Data".Srabotal_Tok_M12;
   "Retain_Data".Timer_Tok_M12_OFF.TON(IN := #_w1 AND ("Unlock_Data".Tok_M12_Real_Temp_Panel < "Retain_Data".Ustavka_tok_M12), PT := T#3s);   // TON coil
   IF #_w1 AND "Retain_Data".Timer_Tok_M12_OFF.Q THEN "Blokirovki_Data".Srabotal_Tok_M12 := FALSE; END_IF;
END_REGION
END_FUNCTION_BLOCK

FUNCTION_BLOCK "Zadanie"   // FB10, LAD
{ S7_Optimized_Access := 'TRUE' }
VERSION : 0.1
   VAR_INPUT
      ValueZad1 : Real;
      ValueZad2 : Real;
      ValueZad3 : Real;
      ValueZad4 : Real;
      ValueZad5 : Real;
      ValueZad6 : Real;
      ValueZad7 : Real;
   END_VAR
   VAR_OUTPUT
      OutAnalog1 : Int;
      OutAnalog2 : Int;
      OutAnalog3 : Int;
      OutAnalog4 : Int;
      OutAnalog5 : Int;
      OutAnalog6 : Int;
      OutAnalog7 : Int;
   END_VAR
   VAR_TEMP
      Soglas1 : Real;
      Soglas2 : Real;
      Soglas3 : Real;
      Soglas4 : Real;
      Soglas5 : Real;
      Soglas6 : Real;
      Soglas7 : Real;
   END_VAR
   VAR CONSTANT
      Constant_1 : Bool;
   END_VAR
BEGIN

REGION Network 1
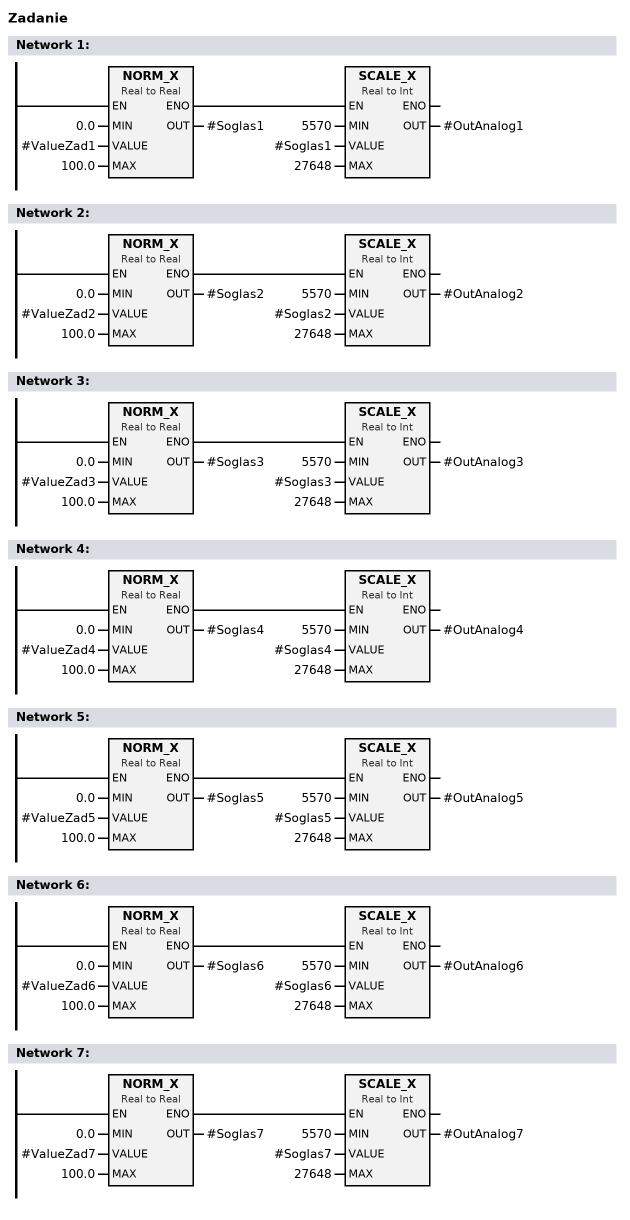
   RUNG wire#powerrail
      { S7_Templates := "[SrcType := Real, DestType := Real]" } Normalize(min := 0.0, value := #ValueZad1, max := 100.0, out => #Soglas1)
      { S7_Templates := "[SrcType := Real, DestType := Int]" } Scale(min := 5570, value := #Soglas1, max := 27648, out => #OutAnalog1)
   END_RUNG
   // the same network as SCL:
   #Soglas1 := NORM_X(MIN := 0.0, VALUE := #ValueZad1, MAX := 100.0);
   #OutAnalog1 := SCALE_X(MIN := 5570, VALUE := #Soglas1, MAX := 27648);
END_REGION

REGION Network 2
   RUNG wire#powerrail
      { S7_Templates := "[SrcType := Real, DestType := Real]" } Normalize(min := 0.0, value := #ValueZad2, max := 100.0, out => #Soglas2)
      { S7_Templates := "[SrcType := Real, DestType := Int]" } Scale(min := 5570, value := #Soglas2, max := 27648, out => #OutAnalog2)
   END_RUNG
   // the same network as SCL:
   #Soglas2 := NORM_X(MIN := 0.0, VALUE := #ValueZad2, MAX := 100.0);
   #OutAnalog2 := SCALE_X(MIN := 5570, VALUE := #Soglas2, MAX := 27648);
END_REGION

REGION Network 3
   RUNG wire#powerrail
      { S7_Templates := "[SrcType := Real, DestType := Real]" } Normalize(min := 0.0, value := #ValueZad3, max := 100.0, out => #Soglas3)
      { S7_Templates := "[SrcType := Real, DestType := Int]" } Scale(min := 5570, value := #Soglas3, max := 27648, out => #OutAnalog3)
   END_RUNG
   // the same network as SCL:
   #Soglas3 := NORM_X(MIN := 0.0, VALUE := #ValueZad3, MAX := 100.0);
   #OutAnalog3 := SCALE_X(MIN := 5570, VALUE := #Soglas3, MAX := 27648);
END_REGION

REGION Network 4
   RUNG wire#powerrail
      { S7_Templates := "[SrcType := Real, DestType := Real]" } Normalize(min := 0.0, value := #ValueZad4, max := 100.0, out => #Soglas4)
      { S7_Templates := "[SrcType := Real, DestType := Int]" } Scale(min := 5570, value := #Soglas4, max := 27648, out => #OutAnalog4)
   END_RUNG
   // the same network as SCL:
   #Soglas4 := NORM_X(MIN := 0.0, VALUE := #ValueZad4, MAX := 100.0);
   #OutAnalog4 := SCALE_X(MIN := 5570, VALUE := #Soglas4, MAX := 27648);
END_REGION

REGION Network 5
   RUNG wire#powerrail
      { S7_Templates := "[SrcType := Real, DestType := Real]" } Normalize(min := 0.0, value := #ValueZad5, max := 100.0, out => #Soglas5)
      { S7_Templates := "[SrcType := Real, DestType := Int]" } Scale(min := 5570, value := #Soglas5, max := 27648, out => #OutAnalog5)
   END_RUNG
   // the same network as SCL:
   #Soglas5 := NORM_X(MIN := 0.0, VALUE := #ValueZad5, MAX := 100.0);
   #OutAnalog5 := SCALE_X(MIN := 5570, VALUE := #Soglas5, MAX := 27648);
END_REGION

REGION Network 6
   RUNG wire#powerrail
      { S7_Templates := "[SrcType := Real, DestType := Real]" } Normalize(min := 0.0, value := #ValueZad6, max := 100.0, out => #Soglas6)
      { S7_Templates := "[SrcType := Real, DestType := Int]" } Scale(min := 5570, value := #Soglas6, max := 27648, out => #OutAnalog6)
   END_RUNG
   // the same network as SCL:
   #Soglas6 := NORM_X(MIN := 0.0, VALUE := #ValueZad6, MAX := 100.0);
   #OutAnalog6 := SCALE_X(MIN := 5570, VALUE := #Soglas6, MAX := 27648);
END_REGION

REGION Network 7
   RUNG wire#powerrail
      { S7_Templates := "[SrcType := Real, DestType := Real]" } Normalize(min := 0.0, value := #ValueZad7, max := 100.0, out => #Soglas7)
      { S7_Templates := "[SrcType := Real, DestType := Int]" } Scale(min := 5570, value := #Soglas7, max := 27648, out => #OutAnalog7)
   END_RUNG
   // the same network as SCL:
   #Soglas7 := NORM_X(MIN := 0.0, VALUE := #ValueZad7, MAX := 100.0);
   #OutAnalog7 := SCALE_X(MIN := 5570, VALUE := #Soglas7, MAX := 27648);
END_REGION
END_FUNCTION_BLOCK

ORGANIZATION_BLOCK "Main"   // OB1, LAD, ProgramCycle
TITLE = "Main Program Sweep (Cycle)"
{ S7_Optimized_Access := 'TRUE' }
VERSION : 0.1
   VAR_INPUT
      Initial_Call : Bool;   // Initial call of this OB
      Remanence : Bool;   // =True, if remanent data are available
   END_VAR
   VAR_TEMP   // added for the SCL form of the ladder/FBD networks
      _w1 : Bool;
   END_VAR
BEGIN

REGION Network 1
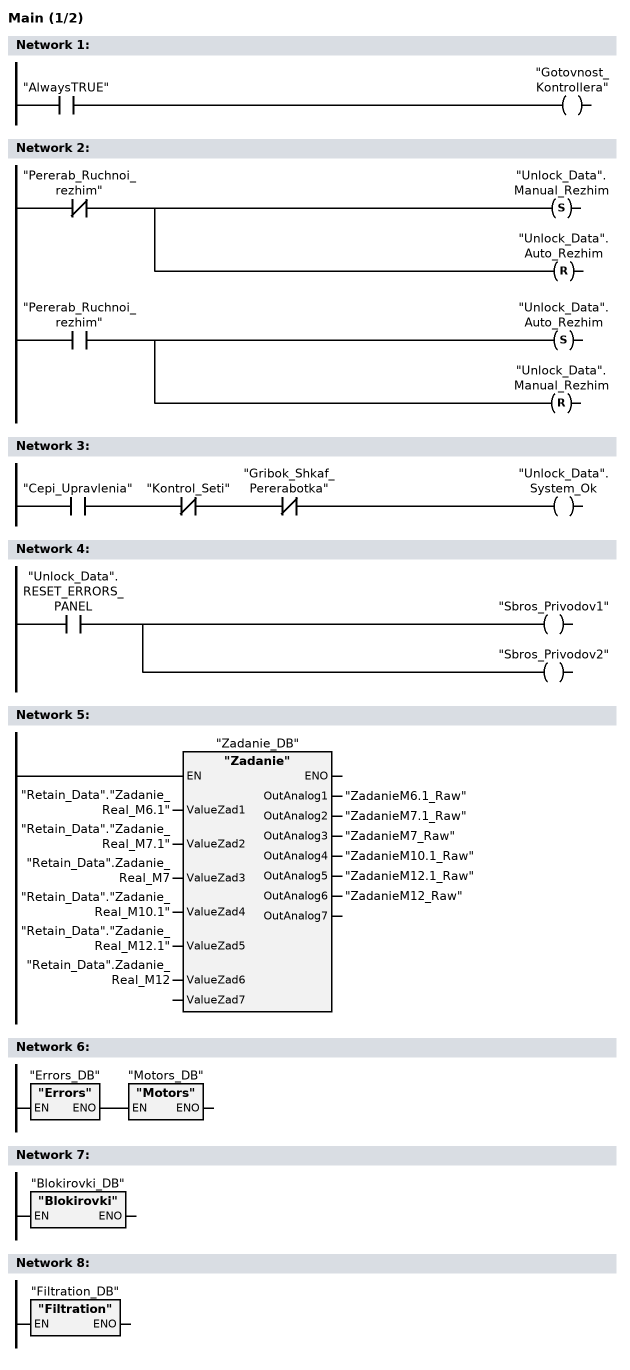
   RUNG wire#powerrail
      Contact( "AlwaysTRUE" )
      Coil( "Gotovnost_Kontrollera" )
   END_RUNG
   // the same network as SCL:
   "Gotovnost_Kontrollera" := "AlwaysTRUE";
END_REGION

REGION Network 2
   RUNG wire#powerrail
      I_Contact( "Pererab_Ruchnoi_rezhim" )
      wire#w1
      S_Coil( "Unlock_Data".Manual_Rezhim )
   END_RUNG
   RUNG wire#w1
      R_Coil( "Unlock_Data".Auto_Rezhim )
   END_RUNG
   RUNG wire#powerrail
      Contact( "Pererab_Ruchnoi_rezhim" )
      wire#w2
      S_Coil( "Unlock_Data".Auto_Rezhim )
   END_RUNG
   RUNG wire#w2
      R_Coil( "Unlock_Data".Manual_Rezhim )
   END_RUNG
   // the same network as SCL:
   IF NOT "Pererab_Ruchnoi_rezhim" THEN
       "Unlock_Data".Manual_Rezhim := TRUE;
       "Unlock_Data".Auto_Rezhim := FALSE;
   END_IF;
   IF "Pererab_Ruchnoi_rezhim" THEN
       "Unlock_Data".Auto_Rezhim := TRUE;
       "Unlock_Data".Manual_Rezhim := FALSE;
   END_IF;
END_REGION

REGION Network 3
   RUNG wire#powerrail
      Contact( "Cepi_Upravlenia" )
      I_Contact( "Kontrol_Seti" )
      I_Contact( "Gribok_Shkaf_Pererabotka" )
      Coil( "Unlock_Data".System_Ok )
   END_RUNG
   // the same network as SCL:
   "Unlock_Data".System_Ok := "Cepi_Upravlenia" AND NOT "Kontrol_Seti" AND NOT "Gribok_Shkaf_Pererabotka";
END_REGION

REGION Network 4
   RUNG wire#powerrail
      Contact( "Unlock_Data".RESET_ERRORS_PANEL )
      wire#w1
      Coil( "Sbros_Privodov1" )
   END_RUNG
   RUNG wire#w1
      Coil( "Sbros_Privodov2" )
   END_RUNG
   // the same network as SCL:
   "Sbros_Privodov1" := "Unlock_Data".RESET_ERRORS_PANEL;
   "Sbros_Privodov2" := "Unlock_Data".RESET_ERRORS_PANEL;
END_REGION

REGION Network 5
   RUNG wire#powerrail
      "Zadanie_DB"(ValueZad1 := "Retain_Data"."Zadanie_Real_M6.1", ValueZad2 := "Retain_Data"."Zadanie_Real_M7.1", ValueZad3 := "Retain_Data".Zadanie_Real_M7, ValueZad4 := "Retain_Data"."Zadanie_Real_M10.1", ValueZad5 := "Retain_Data"."Zadanie_Real_M12.1", ValueZad6 := "Retain_Data".Zadanie_Real_M12, ValueZad7 :=, OutAnalog1 => "ZadanieM6.1_Raw", OutAnalog2 => "ZadanieM7.1_Raw", OutAnalog3 => "ZadanieM7_Raw", OutAnalog4 => "ZadanieM10.1_Raw", OutAnalog5 => "ZadanieM12.1_Raw", OutAnalog6 => "ZadanieM12_Raw", OutAnalog7 =>)
   END_RUNG
   // the same network as SCL:
   "Zadanie_DB"(ValueZad1 := "Retain_Data"."Zadanie_Real_M6.1",   // "Zadanie"
                ValueZad2 := "Retain_Data"."Zadanie_Real_M7.1",
                ValueZad3 := "Retain_Data".Zadanie_Real_M7,
                ValueZad4 := "Retain_Data"."Zadanie_Real_M10.1",
                ValueZad5 := "Retain_Data"."Zadanie_Real_M12.1",
                ValueZad6 := "Retain_Data".Zadanie_Real_M12,
                OutAnalog1 => "ZadanieM6.1_Raw",
                OutAnalog2 => "ZadanieM7.1_Raw",
                OutAnalog3 => "ZadanieM7_Raw",
                OutAnalog4 => "ZadanieM10.1_Raw",
                OutAnalog5 => "ZadanieM12.1_Raw",
                OutAnalog6 => "ZadanieM12_Raw");
END_REGION

REGION Network 6
   RUNG wire#powerrail
      "Errors_DB"()
      "Motors_DB"()
   END_RUNG
   // the same network as SCL:
   "Errors_DB"(ENO => #_w1);   // "Errors"
   IF #_w1 THEN
       "Motors_DB"();   // "Motors"
   END_IF;
END_REGION

REGION Network 7
   RUNG wire#powerrail
      "Blokirovki_DB"()
   END_RUNG
   // the same network as SCL:
   "Blokirovki_DB"();   // "Blokirovki"
END_REGION

REGION Network 8
   RUNG wire#powerrail
      "Filtration_DB"()
   END_RUNG
   // the same network as SCL:
   "Filtration_DB"();   // "Filtration"
END_REGION

REGION Network 9
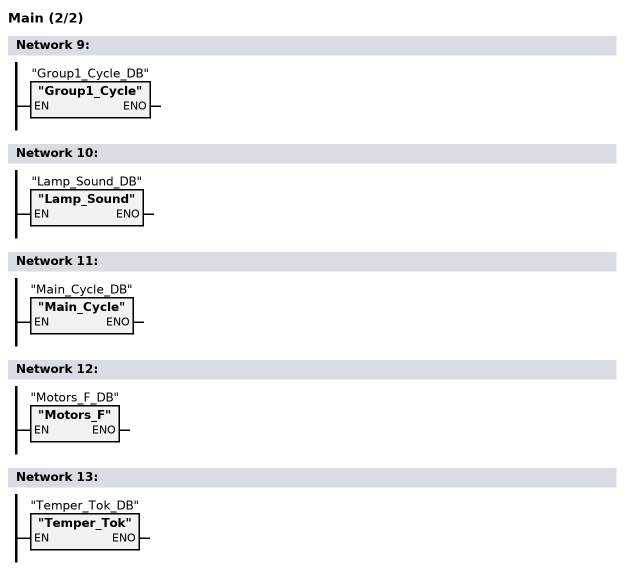
   RUNG wire#powerrail
      "Group1_Cycle_DB"()
   END_RUNG
   // the same network as SCL:
   "Group1_Cycle_DB"();   // "Group1_Cycle"
END_REGION

REGION Network 10
   RUNG wire#powerrail
      "Lamp_Sound_DB"()
   END_RUNG
   // the same network as SCL:
   "Lamp_Sound_DB"();   // "Lamp_Sound"
END_REGION

REGION Network 11
   RUNG wire#powerrail
      "Main_Cycle_DB"()
   END_RUNG
   // the same network as SCL:
   "Main_Cycle_DB"();   // "Main_Cycle"
END_REGION

REGION Network 12
   RUNG wire#powerrail
      "Motors_F_DB"()
   END_RUNG
   // the same network as SCL:
   "Motors_F_DB"();   // "Motors_F"
END_REGION

REGION Network 13
   RUNG wire#powerrail
      "Temper_Tok_DB"()
   END_RUNG
   // the same network as SCL:
   "Temper_Tok_DB"();   // "Temper_Tok"
END_REGION
END_ORGANIZATION_BLOCK

// ===== PLC "PLC_2"  CPU 1214C DC/DC/DC =====

VAR_GLOBAL   // PLC tag table "Default tag table"
   "Tag_2" AT %IW0 : Word;
   "Tag_4" AT %IW8 : Word;
   "Tag_6" AT %IW304 : Word;
   "Tag_8" AT %IW306 : Word;
   "Tag_10" AT %IW308 : Word;
   "Tag_12" AT %IW310 : Word;
   "Tag_14" AT %IW312 : Word;
   "Tag_16" AT %IW314 : Word;
   "Tag_3" AT %QW300 : Word;
   "Tag_5" AT %QW302 : Word;
   "Tag_7" AT %QW0 : Word;
   "Tag_9" AT %QW8 : Word;
   "Tag_11" AT %QW112 : Word;
   "Tag_13" AT %QW114 : Word;
   "Tag_15" AT %QW116 : Word;
   "Tag_17" AT %QW118 : Word;
   "System_Byte" AT %MB1 : Byte;
   "FirstScan" AT %M1.0 : Bool;
   "DiagStatusUpdate" AT %M1.1 : Bool;
   "AlwaysTRUE" AT %M1.2 : Bool;
   "AlwaysFALSE" AT %M1.3 : Bool;
   "Clock_Byte" AT %MB0 : Byte;
   "Clock_10Hz" AT %M0.0 : Bool;
   "Clock_5Hz" AT %M0.1 : Bool;
   "Clock_2.5Hz" AT %M0.2 : Bool;
   "Clock_2Hz" AT %M0.3 : Bool;
   "Clock_1.25Hz" AT %M0.4 : Bool;
   "Clock_1Hz" AT %M0.5 : Bool;
   "Clock_0.625Hz" AT %M0.6 : Bool;
   "Clock_0.5Hz" AT %M0.7 : Bool;
   "Tag_1" AT %M500.0 : Bool;
END_VAR

ORGANIZATION_BLOCK "Main"   // OB1, LAD, ProgramCycle
TITLE = "Main Program Sweep (Cycle)"
{ S7_Optimized_Access := 'TRUE' }
VERSION : 0.1
   VAR_INPUT
      Initial_Call : Bool;   // Initial call of this OB
      Remanence : Bool;   // =True, if remanent data are available
   END_VAR
BEGIN

REGION Network 1
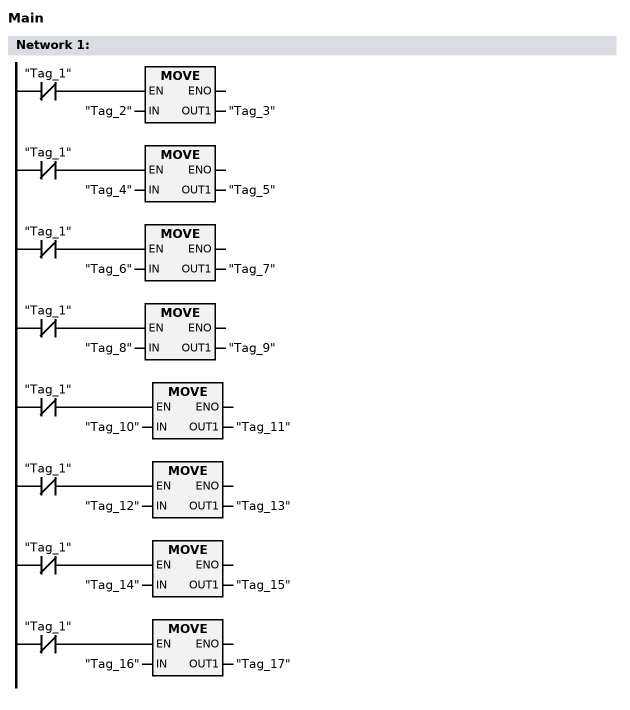
   RUNG wire#powerrail
      I_Contact( "Tag_1" )
      Move(in := "Tag_2", out1 => "Tag_3")
   END_RUNG
   RUNG wire#powerrail
      I_Contact( "Tag_1" )
      Move(in := "Tag_4", out1 => "Tag_5")
   END_RUNG
   RUNG wire#powerrail
      I_Contact( "Tag_1" )
      Move(in := "Tag_6", out1 => "Tag_7")
   END_RUNG
   RUNG wire#powerrail
      I_Contact( "Tag_1" )
      Move(in := "Tag_8", out1 => "Tag_9")
   END_RUNG
   RUNG wire#powerrail
      I_Contact( "Tag_1" )
      Move(in := "Tag_10", out1 => "Tag_11")
   END_RUNG
   RUNG wire#powerrail
      I_Contact( "Tag_1" )
      Move(in := "Tag_12", out1 => "Tag_13")
   END_RUNG
   RUNG wire#powerrail
      I_Contact( "Tag_1" )
      Move(in := "Tag_14", out1 => "Tag_15")
   END_RUNG
   RUNG wire#powerrail
      I_Contact( "Tag_1" )
      Move(in := "Tag_16", out1 => "Tag_17")
   END_RUNG
   // the same network as SCL:
   IF NOT "Tag_1" THEN
       "Tag_3" := "Tag_2";
       "Tag_5" := "Tag_4";
       "Tag_7" := "Tag_6";
       "Tag_9" := "Tag_8";
       "Tag_11" := "Tag_10";
       "Tag_13" := "Tag_12";
       "Tag_15" := "Tag_14";
       "Tag_17" := "Tag_16";
   END_IF;
END_REGION
END_ORGANIZATION_BLOCK

ORGANIZATION_BLOCK "Rack or station failure"   // OB86, LAD, RackStationFailure
{ S7_Optimized_Access := 'TRUE' }
VERSION : 0.1
   VAR_INPUT
      LADDR : Hw_Device;   // Hardware identifier
      Event_Class : Byte;   // Event class
      Fault_ID : Byte;   // Fault identifier
   END_VAR
BEGIN

REGION Network 1
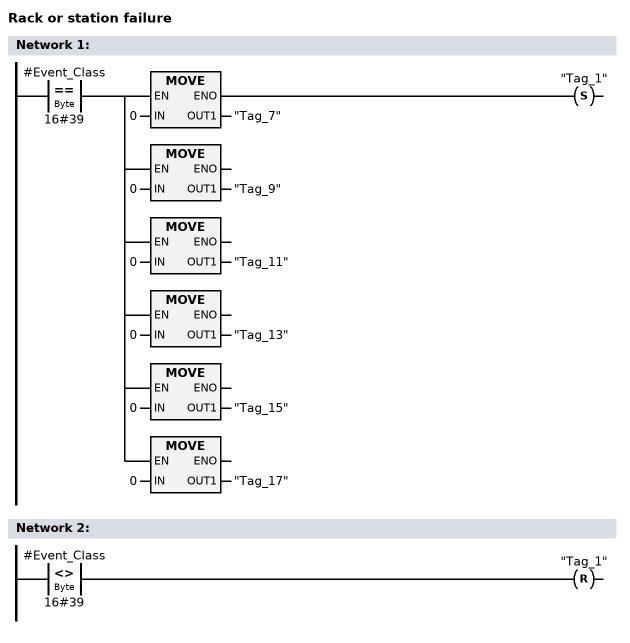
   RUNG wire#powerrail
      { S7_Templates := "SrcType := Byte" } EQ_Contact(in1 := #Event_Class, in2 := 16#39)
      wire#w1
      Move(in := 0, out1 => "Tag_7")
      S_Coil( "Tag_1" )
   END_RUNG
   RUNG wire#w1
      Move(in := 0, out1 => "Tag_9")
   END_RUNG
   RUNG wire#w1
      Move(in := 0, out1 => "Tag_11")
   END_RUNG
   RUNG wire#w1
      Move(in := 0, out1 => "Tag_13")
   END_RUNG
   RUNG wire#w1
      Move(in := 0, out1 => "Tag_15")
   END_RUNG
   RUNG wire#w1
      Move(in := 0, out1 => "Tag_17")
   END_RUNG
   // the same network as SCL:
   IF #Event_Class = 16#39 THEN
       "Tag_7" := 0;
       "Tag_1" := TRUE;
       "Tag_9" := 0;
       "Tag_11" := 0;
       "Tag_13" := 0;
       "Tag_15" := 0;
       "Tag_17" := 0;
   END_IF;
END_REGION

REGION Network 2
   RUNG wire#powerrail
      { S7_Templates := "SrcType := Byte" } NE_Contact(in1 := #Event_Class, in2 := 16#39)
      R_Coil( "Tag_1" )
   END_RUNG
   // the same network as SCL:
   IF #Event_Class <> 16#39 THEN "Tag_1" := FALSE; END_IF;
END_REGION
END_ORGANIZATION_BLOCK